	// Tanks
	{attribute 'OPC.UA.DA' := '1'}
  	{attribute 'OPC.UA.DA.StructuredType' := '1'}
	fbTank_PHUp: 		FB_Tank(TankID:= 'DTK1' ,TankDescr:= 'pH Up Nutrient Tank');
	{attribute 'OPC.UA.DA' := '1'}
  	{attribute 'OPC.UA.DA.StructuredType' := '1'} 
	fbTank_PHDown: 		FB_Tank(TankID:= 'DTK2' ,TankDescr:= 'pH Down Nutrient Tank');
	{attribute 'OPC.UA.DA' := '1'}
  	{attribute 'OPC.UA.DA.StructuredType' := '1'} 
	fbTank_NutrientA: 	FB_Tank(TankID:= 'DTK3' ,TankDescr:= 'Nutrient A Nutrient Tank');
	{attribute 'OPC.UA.DA' := '1'}
  	{attribute 'OPC.UA.DA.StructuredType' := '1'} 
	fbTank_NutrientB: 	FB_Tank(TankID:= 'DTK4' ,TankDescr:= 'Nutrient B Nutrient Tank');
	{attribute 'OPC.UA.DA' := '1'}
  	{attribute 'OPC.UA.DA.StructuredType' := '1'} 
	fbTank_NutrientC: 	FB_Tank(TankID:= 'DTK5' ,TankDescr:= 'Nutrient C Nutrient Tank'); 
	
	{attribute 'OPC.UA.DA' := '1'}
  	{attribute 'OPC.UA.DA.StructuredType' := '1'}
	fbSensor_TankpHUP_LS1: 		FB_Sensor_SICKLevelSwitch_GRF18S(SensorID:= 'DTK1-LS1' , SensorDescr:= 'pH Up Level Switch', 	  SensorType:= E_SensorType.Digital);
	{attribute 'OPC.UA.DA' := '1'}
  	{attribute 'OPC.UA.DA.StructuredType' := '1'}
	fbSensor_TankpHDown_LS1: 	FB_Sensor_SICKLevelSwitch_GRF18S(SensorID:= 'DTK2-LS1' , SensorDescr:= 'pH Down Level Switch', 	  SensorType:= E_SensorType.Digital);
	{attribute 'OPC.UA.DA' := '1'}
  	{attribute 'OPC.UA.DA.StructuredType' := '1'}
	fbSensor_TankNutrientA_LS1: FB_Sensor_SICKLevelSwitch_GRF18S(SensorID:= 'DTK3-LS1' , SensorDescr:= 'Nutrient A Level Switch', SensorType:= E_SensorType.Digital);
	{attribute 'OPC.UA.DA' := '1'}
  	{attribute 'OPC.UA.DA.StructuredType' := '1'}
	fbSensor_TankNutrientB_LS1: FB_Sensor_SICKLevelSwitch_GRF18S(SensorID:= 'DTK4-LS1' , SensorDescr:= 'Nutrient B Level Switch', SensorType:= E_SensorType.Digital);
	{attribute 'OPC.UA.DA' := '1'}
  	{attribute 'OPC.UA.DA.StructuredType' := '1'}
	fbSensor_TankNutrientC_LS1: FB_Sensor_SICKLevelSwitch_GRF18S(SensorID:= 'DTK5-LS1' , SensorDescr:= 'Nutrient C Level Switch', SensorType:= E_SensorType.Digital);
	
	
	// Control Loops
	{attribute 'OPC.UA.DA' := '0'}
	fbControlLoop_Dosing: 		FB_ControlLoop_Dosing(
														DosingPump_phUp := fbDosingPump_phUp, 
														DosingPump_phDOwn := fbDosingPump_phDown, 
														DosingPump_Nutrient_A := fbDosingPump_NutrientA, 
														DosingPump_Nutrient_B := fbDosingPump_NutrientB, 
														DosingPump_Nutrient_C := fbDosingPump_NutrientC, 
														Sensor_EC := fbSensor_EC, 
														Sensor_DO := fbSensor_DissOx, 
														Sensor_ORP := fbSensor_ORP, 
														Sensor_PH := fbSensor_PH, 
														Sensor_TEMP := fbSensor_TMP);
														
	
													
	// Package all components into structure & array 
	// ST used for readability
	// Arrray used for iterability 
	{attribute 'OPC.UA.DA' := '0'}
	stAllComponents: ST_RNDDMComponents;
	
	
	// Interlocks
	{attribute 'OPC.UA.DA' := '1'}
  	{attribute 'OPC.UA.DA.StructuredType' := '1'}
	fbInterlocks: 		FB_InterlockManager;
	
	// Sequences
	{attribute 'OPC.UA.DA' := '0'}
	fbSeqRND_DMMain: 	FB_SequenceRND_Main;
	{attribute 'OPC.UA.DA' := '0'}
	fbSeqRND_DMCal: 	FB_SequenceRND_Calibrate;
	{attribute 'OPC.UA.DA' := '0'}
	fbSeqRND_DMFill: 	FB_SequenceRND_Fill;
	{attribute 'OPC.UA.DA' := '0'}
	aSeqs: ARRAY[1..5] OF FB_SequenceBase;
	
END_VAR

IF GVL.bAutoUpdateDeviceState THEN
	simulation();     // This auto-updates devices eState to the eStateTarget (for testing purposes only)
END_IF

IF bIsFirstRun  THEN
	devices_init();	
	sequence_init();
	bIsFirstRun := FALSE;
END_IF

scanOPCInputs(Inputs := stInputs );
fbSequenceManager(aSequences := aSeqs, fbCurrentSequence := aSeqs[1]);
fbControlLoop_Dosing();

IF GVL.bEnableInterlocks_DM THEN
	interlocks();
END_IF

devices_update();

METHOD checkWaterQuality : BOOL
VAR_INPUT
END_VAR
checkWaterQuality := TRUE;

IF fbSensor_DissOx.getValue() < nDO_Low_Limit OR
	fbSensor_DissOx.getValue() > nDO_High_Limit THEN
	
	checkWaterQuality := FALSE;
	// raise an event
END_IF

IF fbSensor_EC.getValue() < nEC_Low_Limit OR
	fbSensor_EC.getValue() > nEC_High_Limit THEN
	
	checkWaterQuality := FALSE;
	// raise an event
END_IF


IF fbSensor_ORP.getValue() < nORP_Low_Limit OR
	fbSensor_ORP.getValue() > nORP_High_Limit THEN
	
	checkWaterQuality := FALSE;
	// raise an event
END_IF


IF fbSensor_PH.getValue() < nPH_Low_Limit OR
	fbSensor_PH.getValue() > nPH_High_Limit THEN
	
	checkWaterQuality := FALSE;
	// raise an event
END_IF


IF fbSensor_TMP.getValue() < nTemp_Low_Limit OR
	fbSensor_TMP.getValue() > nTemp_High_Limit THEN
	
	checkWaterQuality := FALSE;
	// raise an event
END_IF
END_METHOD

METHOD devices_init : BOOL
VAR
	VarInfo : __SYSTEM.VAR_INFO;
END_VAR
// Hold References to devices in a structure and also an array
// A structure is useful where devices are accessed by name (handy with auto-complete and readability)
// The array is useful for when we want to iterate through all of the devices in the machine and apply a global command (i.e. disable all devices)

// Add physical entity sensors to physical entities (i.e. tanks)
fbSumpDosing.fbSensor_H := fbSensor_SumpLSH;
fbSumpDosing.bSensorH_Enable := TRUE;

fbTank_PHUp.fbSensor_H := fbSensor_TankpHUP_LS1;
fbTank_PHUp.bSensorH_Enable := TRUE;

fbTank_PHDown.fbSensor_H := fbSensor_TankpHDown_LS1;
fbTank_PHDown.bSensorH_Enable := TRUE;

fbTank_NutrientA.fbSensor_H := fbSensor_TankNutrientA_LS1;
fbTank_NutrientA.bSensorH_Enable := TRUE;

fbTank_NutrientB.fbSensor_H := fbSensor_TankNutrientB_LS1;
fbTank_NutrientB.bSensorH_Enable := TRUE;

fbTank_NutrientC.fbSensor_H := fbSensor_TankNutrientC_LS1;
fbTank_NutrientC.bSensorH_Enable := TRUE;

// Extract the function block instance name and insert it to each function block
// This enables us to share only the function block name over OPC for nested instances (i.e. sequences, interlock manager)
// The contents of each function block is shared over OPC within the Machine as per heirarchy
// When Ignition needs to retrieve details of devices at the interlock manager and sequence, it simply performs a lookup using the VarID as a key


VarInfo := __VARINFO(fbControlLoop_Dosing);
fbControlLoop_Dosing.setVarID(VarID := VarInfo.Symbol);

VarInfo := __VARINFO(fbDosingPump_NutrientA);
fbDosingPump_NutrientA.setVarID(VarID := VarInfo.Symbol);

VarInfo := __VARINFO(fbDosingPump_NutrientB);
fbDosingPump_NutrientB.setVarID(VarID := VarInfo.Symbol);

VarInfo := __VARINFO(fbDosingPump_NutrientC);
fbDosingPump_NutrientC.setVarID(VarID := VarInfo.Symbol);

VarInfo := __VARINFO(fbDosingPump_phDown);
fbDosingPump_phDown.setVarID(VarID := VarInfo.Symbol);

VarInfo := __VARINFO(fbDosingPump_phUp);
fbDosingPump_phUp.setVarID(VarID := VarInfo.Symbol);

VarInfo := __VARINFO(fbPump_MainPumpA);
fbPump_MainPumpA.setVarID(VarID := VarInfo.Symbol);

VarInfo := __VARINFO(fbSensor_DissOx);
fbSensor_DissOx.setVarID(VarID := VarInfo.Symbol);

VarInfo := __VARINFO(fbSensor_DosingPIT1);
fbSensor_DosingPIT1.setVarID(VarID := VarInfo.Symbol);

VarInfo := __VARINFO(fbSensor_EC);
fbSensor_EC.setVarID(VarID := VarInfo.Symbol);

VarInfo := __VARINFO(fbSensor_FilterPIT1);
fbSensor_FilterPIT1.setVarID(VarID := VarInfo.Symbol);

VarInfo := __VARINFO(fbSensor_FilterPIT2);
fbSensor_FilterPIT2.setVarID(VarID := VarInfo.Symbol);

VarInfo := __VARINFO(fbSensor_ORP);
fbSensor_ORP.setVarID(VarID := VarInfo.Symbol);

VarInfo := __VARINFO(fbSensor_PH);
fbSensor_PH.setVarID(VarID := VarInfo.Symbol);

VarInfo := __VARINFO(fbSensor_SumpLSH );
fbSensor_SumpLSH .setVarID(VarID := VarInfo.Symbol);

VarInfo := __VARINFO(fbSensor_TankNutrientA_LS1);
fbSensor_TankNutrientA_LS1.setVarID(VarID := VarInfo.Symbol);

VarInfo := __VARINFO(fbSensor_TankNutrientB_LS1);
fbSensor_TankNutrientB_LS1.setVarID(VarID := VarInfo.Symbol);

VarInfo := __VARINFO(fbSensor_TankNutrientC_LS1);
fbSensor_TankNutrientC_LS1.setVarID(VarID := VarInfo.Symbol);

VarInfo := __VARINFO(fbSensor_TankpHDown_LS1);
fbSensor_TankpHDown_LS1.setVarID(VarID := VarInfo.Symbol);

VarInfo := __VARINFO(fbSensor_TankpHUP_LS1);
fbSensor_TankpHUP_LS1.setVarID(VarID := VarInfo.Symbol);

VarInfo := __VARINFO(fbSensor_TMP);
fbSensor_TMP.setVarID(VarID := VarInfo.Symbol);

VarInfo := __VARINFO(fbSumpDosing);
fbSumpDosing.setVarID(VarID := VarInfo.Symbol);

VarInfo := __VARINFO(fbTank_NutrientA);
fbTank_NutrientA.setVarID(VarID := VarInfo.Symbol);

VarInfo := __VARINFO(fbTank_NutrientB);
fbTank_NutrientB.setVarID(VarID := VarInfo.Symbol);

VarInfo := __VARINFO(fbTank_NutrientC);
fbTank_NutrientC.setVarID(VarID := VarInfo.Symbol);

VarInfo := __VARINFO(fbTank_PHDown);
fbTank_PHDown.setVarID(VarID := VarInfo.Symbol);

VarInfo := __VARINFO(fbTank_PHUp);
fbTank_PHUp.setVarID(VarID := VarInfo.Symbol);

VarInfo := __VARINFO(fbUVFilter1);
fbUVFilter1.setVarID(VarID := VarInfo.Symbol);

VarInfo := __VARINFO(fbValve_IrrigatorSupply);
fbValve_IrrigatorSupply.setVarID(VarID := VarInfo.Symbol);

VarInfo := __VARINFO(fbValve_RevOsSupply);
fbValve_RevOsSupply.setVarID(VarID := VarInfo.Symbol);


aAllComponents[1]  :=  ADR(fbSensor_DissOx );
aAllComponents[2]  :=  ADR(fbSensor_EC );
aAllComponents[3]  :=  ADR(fbSensor_ORP );
aAllComponents[4]  :=  ADR(fbSensor_PH );
aAllComponents[5]  :=  ADR(fbSensor_TMP );
aAllComponents[6]  :=  ADR(fbSensor_SumpLSH  );
aAllComponents[7]  :=  ADR(fbSensor_FilterPIT1 );
aAllComponents[8]  :=  ADR(fbSensor_FilterPIT2 );
aAllComponents[9]  :=  ADR(fbSensor_DosingPIT1 );
aAllComponents[10]  :=  ADR(fbDosingPump_phUp );
aAllComponents[11]  :=  ADR(fbDosingPump_phDown );
aAllComponents[12]  :=  ADR(fbDosingPump_NutrientA );
aAllComponents[13]  :=  ADR(fbDosingPump_NutrientB );
aAllComponents[14]  :=  ADR(fbDosingPump_NutrientC );
aAllComponents[15]  :=  ADR(fbValve_RevOsSupply );
aAllComponents[16]  :=  ADR(fbValve_IrrigatorSupply );
aAllComponents[17]  :=  ADR(fbPump_MainPumpA);
aAllComponents[18]  :=  ADR(fbUVFilter1 );
aAllComponents[19]  :=  ADR(fbSumpDosing );
aAllComponents[20]  :=  ADR(fbTank_PHUp );
aAllComponents[21]  :=  ADR(fbTank_PHDown );
aAllComponents[22]  :=  ADR(fbTank_NutrientA );
aAllComponents[23]  :=  ADR(fbTank_NutrientB );
aAllComponents[24]  :=  ADR(fbTank_NutrientC );
aAllComponents[25]  :=  ADR(fbSensor_TankpHUP_LS1 );
aAllComponents[26]  :=  ADR(fbSensor_TankpHDown_LS1 );
aAllComponents[27]  :=  ADR(fbSensor_TankNutrientA_LS1 );
aAllComponents[28]  :=  ADR(fbSensor_TankNutrientB_LS1 );
aAllComponents[29]  :=  ADR(fbSensor_TankNutrientC_LS1 );


stAllComponents.fbValve_RevOsSupply  := ADR(fbValve_RevOsSupply);
stAllComponents.fbValve_IrrigatorSupply  := ADR(fbValve_IrrigatorSupply);
stAllComponents.fbPump_MainPumpA  := ADR(fbPump_MainPumpA);
stAllComponents.fbUVFilter1  := ADR(fbUVFilter1);
stAllComponents.fbSumpDosing  := ADR(fbSumpDosing);
stAllComponents.fbDosingPump_phUp  := ADR(fbDosingPump_phUp);
stAllComponents.fbDosingPump_phDown  := ADR(fbDosingPump_phDown);
stAllComponents.fbDosingPump_NutrientA  := ADR(fbDosingPump_NutrientA);
stAllComponents.fbDosingPump_NutrientB  := ADR(fbDosingPump_NutrientB);
stAllComponents.fbDosingPump_NutrientC  := ADR(fbDosingPump_NutrientC);
stAllComponents.fbSensor_DissOx1  := ADR(fbSensor_DissOx);
stAllComponents.fbSensor_EC1  := ADR(fbSensor_EC);
stAllComponents.fbSensor_ORP1  := ADR(fbSensor_ORP);
stAllComponents.fbSensor_PH1  := ADR(fbSensor_PH);
stAllComponents.fbSensor_TMP1  := ADR(fbSensor_TMP);
stAllComponents.fbSensor_SumpLSH  := ADR(fbSensor_SumpLSH);
stAllComponents.fbSensor_TankpHUP_LS1  := ADR(fbSensor_TankpHUP_LS1);
stAllComponents.fbSensor_TankpHDown_LS1  := ADR(fbSensor_TankpHDown_LS1);
stAllComponents.fbSensor_TankNutrientA_LS1  := ADR(fbSensor_TankNutrientA_LS1);
stAllComponents.fbSensor_TankNutrientB_LS1  := ADR(fbSensor_TankNutrientB_LS1);
stAllComponents.fbSensor_TankNutrientC_LS1  := ADR(fbSensor_TankNutrientC_LS1);
stAllComponents.fbSensor_FilterPIT1  := ADR(fbSensor_FilterPIT1);
stAllComponents.fbSensor_FilterPIT2  := ADR(fbSensor_FilterPIT2);
stAllComponents.fbSensor_DosingPIT1  := ADR(fbSensor_DosingPIT1);
stAllComponents.fbTank_pHUP  := ADR(fbTank_pHUP);
stAllComponents.fbTank_pHDown  := ADR(fbTank_pHDown);
stAllComponents.fbTank_NutrientA  := ADR(fbTank_NutrientA);
stAllComponents.fbTank_NutrientB  := ADR(fbTank_NutrientB);
stAllComponents.fbTank_NutrientC  := ADR(fbTank_NutrientC);
stAllComponents.fbControlLoop_Dosing  := ADR(fbControlLoop_Dosing);

nQtyComponents := 29;

devices_disable_All();
END_METHOD

METHOD devices_update : BOOL
VAR_INPUT
END_VAR
fbModbusMaster();
fbDosingPump_phUp(fbModbusMaster := fbModbusMaster);
fbDosingPump_phDown(fbModbusMaster := fbModbusMaster);
fbDosingPump_NutrientA(fbModbusMaster := fbModbusMaster);
fbDosingPump_NutrientB(fbModbusMaster := fbModbusMaster);
fbDosingPump_NutrientC(fbModbusMaster := fbModbusMaster);
fbSensor_DissOx();
fbSensor_EC();
fbSensor_ORP();
fbSensor_PH();
fbSensor_TMP();
fbSensor_SumpLSH ();
fbSensor_FilterPIT1();
fbSensor_FilterPIT2();
fbSensor_DosingPIT1();
fbValve_RevOsSupply();
fbValve_IrrigatorSupply();
fbPump_MainPumpA();
fbUVFilter1();
fbSumpDosing();
fbTank_PHUp();
fbTank_PHDown();
fbTank_NutrientA();
fbTank_NutrientB();
fbTank_NutrientC();
fbSensor_TankpHUP_LS1();
fbSensor_TankpHDown_LS1();
fbSensor_TankNutrientA_LS1();
fbSensor_TankNutrientB_LS1();
fbSensor_TankNutrientC_LS1();
fbControlLoop_Dosing();
END_METHOD

METHOD FB_init : BOOL
VAR_INPUT
	bInitRetains : BOOL; // if TRUE, the retain variables are initialized (warm start / cold start)
	bInCopyCode : BOOL;  // if TRUE, the instance afterwards gets moved into the copy code (online change)
	
	ID: STRING;
	Description: STRING;
	//Pump_ModbusID: INT;
END_VAR
sID := ID;
sDescr := Description;
//nAgrowtekModbusID := Pump_ModbusID;
END_METHOD

METHOD interlocks : BOOL
VAR_INPUT
END_VAR
fbInterlocks.init();

fbInterlocks.update(
							Description:= 'Nutrient B Dosing Pump - RUNNING',
							InterlockType:= E_InterlockType.RunInterlock, 
							Subject_Device:= ADR(fbDosingPump_NutrientA), 
							Subject_State:= E_DeviceState.IDLE, 
							Signal:= E_DeviceState.RUNNING = fbDosingPump_NutrientB.getState(), 
							HoldSequence:=	TRUE );
				
							
fbInterlocks.update(
							Description:= 'Nutrient C Dosing Pump - RUNNING',
							InterlockType:= E_InterlockType.RunInterlock, 
							Subject_Device:= ADR(fbDosingPump_NutrientA), 
							Subject_State:= E_DeviceState.IDLE, 
							Signal:= fbDosingPump_NutrientC.getState() = E_DeviceState.RUNNING, 
							HoldSequence:=	TRUE );
							
fbInterlocks.update(
							Description:= 'PH Down Dosing Pump - RUNNING',
							InterlockType:= E_InterlockType.RunInterlock, 
							Subject_Device:= ADR(fbDosingPump_NutrientA), 
							Subject_State:= E_DeviceState.IDLE, 
							Signal := fbDosingPump_phDown.getState() = E_DeviceState.RUNNING, 
							HoldSequence:=	TRUE );
							
fbInterlocks.update(
							Description:= 'PH Up Dosing Pump - RUNNING',
							InterlockType:= E_InterlockType.RunInterlock, 
							Subject_Device:= ADR(fbDosingPump_NutrientA), 
							Subject_State:= E_DeviceState.IDLE, 
							Signal := fbDosingPump_phUp.getState() = E_DeviceState.RUNNING, 
							HoldSequence:=	TRUE );
								
							
fbInterlocks.update(
							Description:= 'Dosing Line Pressure - OUT OF RANGE',
							InterlockType:= E_InterlockType.RunInterlock, 
							Subject_Device:= ADR(fbDosingPump_NutrientA), 
							Subject_State:= E_DeviceState.IDLE, 
							Signal:= fbSensor_DosingPIT1.getState() = E_DeviceState.OUT_OF_RANGE, 
							HoldSequence:=	FALSE );
							
							
// Dosing Pump - Nutrient B Interlocks

fbInterlocks.update(
							Description:= 'Nutrient A Dosing Pump - RUNNING',
							InterlockType:= E_InterlockType.RunInterlock, 
							Subject_Device:= ADR(fbDosingPump_NutrientB), 
							Subject_State:= E_DeviceState.IDLE, 
							Signal:= fbDosingPump_NutrientA.getState() = E_DeviceState.RUNNING, 
							HoldSequence:=	TRUE );
							
fbInterlocks.update(
							Description:= 'Nutrient B Dosing Pump - RUNNING',
							InterlockType:= E_InterlockType.RunInterlock, 
							Subject_Device:= ADR(fbDosingPump_NutrientB), 
							Subject_State:= E_DeviceState.IDLE, 
							Signal := fbDosingPump_NutrientC.getState() = E_DeviceState.RUNNING, 
							HoldSequence:=	TRUE );
							
fbInterlocks.update(
							Description:= 'PH Down Dosing Pump - RUNNING',
							InterlockType:= E_InterlockType.RunInterlock, 
							Subject_Device:= ADR(fbDosingPump_NutrientB), 
							Subject_State:= E_DeviceState.IDLE, 
							Signal:= fbDosingPump_phDown.getState() = E_DeviceState.RUNNING, 
							HoldSequence:=	TRUE );
							
fbInterlocks.update(
							Description:= 'PH Up Dosing Pump - RUNNING',	
							InterlockType:= E_InterlockType.RunInterlock, 
							Subject_Device:= ADR(fbDosingPump_NutrientB), 
							Subject_State:= E_DeviceState.IDLE, 
							Signal:= fbDosingPump_phUp.getState() = E_DeviceState.RUNNING, 
							HoldSequence:=	TRUE );
							

							
fbInterlocks.update(
							Description:= 'Dosing Line Pressure - OUT OF RANGE',
							InterlockType:= E_InterlockType.RunInterlock, 
							Subject_Device:= ADR(fbDosingPump_NutrientB), 
							Subject_State:= E_DeviceState.IDLE, 
							Signal:= fbSensor_DosingPIT1.getState() = E_DeviceState.OUT_OF_RANGE, 
							HoldSequence:=	FALSE );

							
// Dosing Pump - Nutrient C Interlocks

fbInterlocks.update(
							Description:= 'Nutrient A Dosing Pump - RUNNING',
							InterlockType:= E_InterlockType.RunInterlock, 
							Subject_Device:= ADR(fbDosingPump_NutrientC), 
							Subject_State:= E_DeviceState.IDLE, 
							Signal:= fbDosingPump_NutrientA.getState() = E_DeviceState.RUNNING, 
							HoldSequence:=	TRUE );
							
fbInterlocks.update(
							Description:= 'Nutrient B Dosing Pump - RUNNING',
							InterlockType:= E_InterlockType.RunInterlock, 
							Subject_Device:= ADR(fbDosingPump_NutrientC), 
							Subject_State:= E_DeviceState.IDLE, 
							Signal:= fbDosingPump_NutrientB.getState() = E_DeviceState.RUNNING, 
							HoldSequence:=	TRUE );
							
fbInterlocks.update(
							Description:= 'PH Down Dosing Pump - RUNNING',	
							InterlockType:= E_InterlockType.RunInterlock, 
							Subject_Device:= ADR(fbDosingPump_NutrientC), 
							Subject_State:= E_DeviceState.IDLE, 
							Signal:= fbDosingPump_phDown.getState() = E_DeviceState.RUNNING, 
							HoldSequence:=	TRUE );
							
fbInterlocks.update(
							Description:= 'PH Up Dosing Pump - RUNNING',	
							InterlockType:= E_InterlockType.RunInterlock, 
							Subject_Device:= ADR(fbDosingPump_NutrientC), 
							Subject_State:= E_DeviceState.IDLE, 
							Signal:= fbDosingPump_phUp.getState() = E_DeviceState.RUNNING, 
							HoldSequence:=	TRUE );
							
							
fbInterlocks.update(
							Description:= 'Dosing Line Pressure - OUT OF RANGE',
							InterlockType:= E_InterlockType.StartPermissive, 
							Subject_Device:= ADR(fbDosingPump_NutrientC), 
							Subject_State:= E_DeviceState.IDLE, 
							Signal:= fbSensor_DosingPIT1.getState() = E_DeviceState.OUT_OF_RANGE, 
							HoldSequence:=	FALSE );
							
							
// Dosing Pump - PH Up Interlocks
fbInterlocks.update(
							Description:= 'Nutrient A Dosing Pump - RUNNING',	
							InterlockType:= E_InterlockType.RunInterlock, 
							Subject_Device:= ADR(fbDosingPump_phUp), 
							Subject_State:= E_DeviceState.IDLE, 
							Signal:= fbDosingPump_NutrientA.getState() = E_DeviceState.RUNNING, 
							HoldSequence:=	TRUE );
							
fbInterlocks.update(
							Description:= 'Nutrient B Dosing Pump - RUNNING',	
							InterlockType:= E_InterlockType.RunInterlock, 
							Subject_Device:= ADR(fbDosingPump_phUp), 
							Subject_State:= E_DeviceState.IDLE, 
							Signal:= fbDosingPump_NutrientB.getState() = E_DeviceState.RUNNING, 
							HoldSequence:=	TRUE );
							
fbInterlocks.update(
							Description:= 'Nutrient C Dosing Pump - RUNNING',
							InterlockType:= E_InterlockType.RunInterlock, 
							Subject_Device:= ADR(fbDosingPump_phUp), 
							Subject_State:= E_DeviceState.IDLE, 
							Signal:= fbDosingPump_NutrientC.getState() = E_DeviceState.RUNNING, 
							HoldSequence:=	TRUE );
							
fbInterlocks.update(
							Description:= 'PH Down Dosing Pump - RUNNING',
							InterlockType:= E_InterlockType.RunInterlock, 
							Subject_Device:= ADR(fbDosingPump_phUp), 
							Subject_State:= E_DeviceState.IDLE, 
							Signal:= fbDosingPump_phDown.getState() = E_DeviceState.RUNNING, 
							HoldSequence:=	TRUE );
					
							
fbInterlocks.update(
							Description:= 'Dosing Line Pressure - OUT OF RANGE',		
							InterlockType:= E_InterlockType.StartPermissive, 
							Subject_Device:= ADR(fbDosingPump_phUp), 
							Subject_State:= E_DeviceState.IDLE, 
							Signal:= fbSensor_DosingPIT1.getState() = E_DeviceState.OUT_OF_RANGE, 
							HoldSequence:=	FALSE );	
						
							
// Dosing Pump - PH Down Interlocks
fbInterlocks.update(
							Description:= 'Nutrient A Dosing Pump - RUNNING',		
							InterlockType:= E_InterlockType.RunInterlock, 
							Subject_Device:= ADR(fbDosingPump_phDown), 
							Subject_State:= E_DeviceState.IDLE, 
							Signal:= fbDosingPump_NutrientA.getState() = E_DeviceState.RUNNING, 
							HoldSequence:=	TRUE );
							
fbInterlocks.update(
							Description:= 'Nutrient B Dosing Pump - RUNNING',	
							InterlockType:= E_InterlockType.RunInterlock, 
							Subject_Device:= ADR(fbDosingPump_phDown), 
							Subject_State:= E_DeviceState.IDLE, 
							Signal:= fbDosingPump_NutrientB.getState() = E_DeviceState.RUNNING, 
							HoldSequence:=	TRUE );
							
fbInterlocks.update(
							Description:= 'Nutrient C Dosing Pump - RUNNING',	
							InterlockType:= E_InterlockType.RunInterlock, 
							Subject_Device:= ADR(fbDosingPump_phDown), 
							Subject_State:= E_DeviceState.IDLE, 
							Signal:= fbDosingPump_NutrientC.getState() = E_DeviceState.RUNNING, 
							HoldSequence:=	TRUE );
							
fbInterlocks.update(
							Description:= 'PH Up Dosing Pump - RUNNING',		
							InterlockType:= E_InterlockType.RunInterlock, 
							Subject_Device:= ADR(fbDosingPump_phDown), 
							Subject_State:= E_DeviceState.IDLE, 
							Signal:= fbDosingPump_phUp.getState() = E_DeviceState.RUNNING, 
							HoldSequence:=	TRUE );
							
fbInterlocks.update(
							Description:= 'Dosing Line Pressure - OUT OF RANGE',		
							InterlockType:= E_InterlockType.RunInterlock, 
							Subject_Device:= ADR(fbDosingPump_phDown), 
							Subject_State:= E_DeviceState.IDLE, 
							Signal:= fbSensor_DosingPIT1.getState() = E_DeviceState.OUT_OF_RANGE, 
							HoldSequence:=	FALSE );

							
// Main Pump A - Interlocks	
fbInterlocks.update(
							Description:= 'Dosing Sump - LOW LOW Level',	
							InterlockType:= E_InterlockType.RunInterlock, 
							Subject_Device:= ADR(fbPump_MainPumpA), 
							Subject_State:= E_DeviceState.IDLE, 
							Signal:= fbSumpDosing.getState() = E_DeviceState.LOW_LOW,
							HoldSequence:=	TRUE );	
										

							
							
							
fbInterlocks.update(
							Description:= 'Bag Filter 1 - OVER-PRESSURE',
							InterlockType:= E_InterlockType.RunInterlock, 
							Subject_Device:= ADR(fbPump_MainPumpA), 
							Subject_State:= E_DeviceState.IDLE, 
							Signal:= (fbSensor_FilterPIT2.getValue() - fbSensor_FilterPIT1.getValue())  > nBagFilterPressureMax,
							HoldSequence:=	TRUE ); 
							
fbInterlocks.update(
							Description:= 'Bag Filter 2 - OVER-PRESSURE',
							InterlockType:= E_InterlockType.RunInterlock, 
							Subject_Device:= ADR(fbPump_MainPumpA), 
							Subject_State:= E_DeviceState.IDLE, 
							Signal:= (fbSensor_DosingPIT1.getValue() - fbSensor_FilterPIT2.getValue()  > nBagFilterPressureMax),
							HoldSequence:=	TRUE );
	
							
// UV Filter - Interlocks					

fbInterlocks.update(
							Description:= 'Dosing Line - Low Pressure',
							InterlockType:= E_InterlockType.RunInterlock, 
							Subject_Device:= ADR(fbUVFilter1), 
							Subject_State:= E_DeviceState.OFF, 
							Signal:= fbSensor_DosingPIT1.getValue() < nPressureMin_Dosing, 
							HoldSequence:=	TRUE );	

// Valve - Irrigator Supply				

fbInterlocks.update(
							Description:= 'Water Quality (EC,pH,ORP,DO and temp) - OUT OF RANGE',
							InterlockType:= E_InterlockType.RunInterlock, 
							Subject_Device:= ADR(fbValve_IrrigatorSupply), 
							Subject_State:= E_DeviceState.CLOSED, 
							Signal:= checkWaterQuality(), 
							HoldSequence:=	TRUE );			
							
fbInterlocks.execute();
END_METHOD

METHOD scanOPCInputs : BOOL
VAR_INPUT
	Inputs: ST_INPUTS_RND_DosingMachine;
END_VAR

(*
			SEQUENCE CONTROL
*)



IF stInputs.stSequenceManager.Sequence_Selected <> fbSequenceManager.getCurrentSeq_ID() THEN // Selected sequence has been changed
	fbSequenceManager.stopSequence();
	devices_disable_All();
	fbSequenceManager.selectSequence(stInputs.stSequenceManager.Sequence_Selected);
	devices_enable_CurrSeq();
	//fbSequenceManager.startSequence(); // Automatically start sequence on change of sequence selected - can change this if required
END_IF


IF stInputs.stSequenceManager.Sequence_Ack_Interlock THEN
	fbSequenceManager.acknowledgePause();
	stInputs.stSequenceManager.Sequence_Ack_Interlock := FALSE;
END_IF



CASE stInputs.stSequenceManager.Sequence_Command OF
	E_SequenceState.RUN:
		IF fbSequenceManager.getState() <> E_SequenceState.RUN THEN
			fbSequenceManager.startSequence();
			stInputs.stSequenceManager.Sequence_Command := E_SequenceState.WAIT;
		END_IF
	E_SequenceState.STOP:
		IF fbSequenceManager.getState() <> E_SequenceState.STOP THEN
			fbSequenceManager.stopSequence();
			stInputs.stSequenceManager.Sequence_Command := E_SequenceState.WAIT;
		END_IF
	E_SequenceState.HOLD:
		IF fbSequenceManager.getState() <> E_SequenceState.HOLD THEN
			fbSequenceManager.pauseSequence();
			stInputs.stSequenceManager.Sequence_Command := E_SequenceState.WAIT;
		END_IF
END_CASE


(*
			WATER QUALITY LIMITS
*)


nEC_Low_Limit := stInputs.stWaterQuality.EC_LOW_Limit;
nEC_High_Limit := stInputs.stWaterQuality.EC_HIGH_Limit;
nEC_SetPoint := stInputs.stWaterQuality.EC_SetPoint;

nPH_Low_Limit := stInputs.stWaterQuality.PH_LOW_Limit;
nPH_High_Limit := stInputs.stWaterQuality.PH_HIGH_Limit;
nPH_SetPoint := stInputs.stWaterQuality.PH_SetPoint;

nDO_Low_Limit := stInputs.stWaterQuality.DO_LOW_Limit;
nDO_High_Limit := stInputs.stWaterQuality.DO_HIGH_Limit;
nDO_SetPoint := stInputs.stWaterQuality.DO_SetPoint;

nORP_Low_Limit := stInputs.stWaterQuality.ORP_LOW_Limit;
nORP_High_Limit := stInputs.stWaterQuality.ORP_HIGH_Limit;
nORP_SetPoint := stInputs.stWaterQuality.ORP_SetPoint;

nTemp_Low_Limit := stInputs.stWaterQuality.Temp_LOW_Limit;
nTemp_Low_Limit := stInputs.stWaterQuality.Temp_LOW_Limit;
nTemp_SetPoint := stInputs.stWaterQuality.Temp_SetPoint;

(*
			PRESSURE LIMITS
*)

//nPressureMin_Dosing := stInputs.Dosing_Pressure_LOW_Limit;
//nPressureMax_Dosing := stInputs.Dosing_Pressure_HIGH_Limit;


(*
			ACTUATORS
*)

fbValve_IrrigatorSupply.setMode(Mode := stInputs.stValve_IrrigatorSupply.Mode);
IF fbValve_IrrigatorSupply.inManual() THEN
	fbValve_IrrigatorSupply.setCommand(StateTarget := stInputs.stValve_IrrigatorSupply.Command);
END_IF

fbUVFilter1.setMode(Mode := stInputs.stUVFilter.Mode);
IF fbUVFilter1.inManual() THEN
	fbUVFilter1.setCommand(StateTarget := stInputs.stUVFilter.Command);
END_IF

// Dosing Pump - PH UP
fbDosingPump_phUp.setMode(Mode := stInputs.stDosingPump_phUp.Mode);
IF fbDosingPump_phUp.inManual() THEN
	fbDosingPump_phUp.setCommand(StateTarget := stInputs.stDosingPump_phUp.Command);
END_IF
						
// Dosing Pump - PH Down
fbDosingPump_phDown.setMode(Mode := stInputs.stDosingPump_phDown.Mode);
IF fbDosingPump_phDown.inManual() THEN
	fbDosingPump_phDown.setCommand(StateTarget := stInputs.stDosingPump_phDown.Command);
END_IF

// Dosing Pump - Nutrient A
fbDosingPump_NutrientA.setMode(Mode := stInputs.stDosingPump_NutrientA.Mode);
IF fbDosingPump_NutrientA.inManual() THEN
	fbDosingPump_NutrientA.setCommand(StateTarget := stInputs.stDosingPump_NutrientA.Command);
END_IF

// Dosing Pump - Nutrient B
fbDosingPump_NutrientB.setMode(Mode := stInputs.stDosingPump_NutrientB.Mode);
IF fbDosingPump_NutrientB.inManual() THEN
	fbDosingPump_NutrientB.setCommand(StateTarget := stInputs.stDosingPump_NutrientB.Command);
END_IF

// Dosing Pump - Nutrient C
fbDosingPump_NutrientC.setMode(Mode := stInputs.stDosingPump_NutrientC.Mode);
IF fbDosingPump_NutrientC.inManual() THEN
	fbDosingPump_NutrientC.setCommand(StateTarget := stInputs.stDosingPump_NutrientC.Command);
END_IF
						

// Main Pump A
fbPump_MainPumpA.setMode(Mode := stInputs.stPump_MainPumpA.Mode);
IF fbPump_MainPumpA.inManual() THEN
	fbPump_MainPumpA.setCommand(StateTarget := stInputs.stPump_MainPumpA.Command);
END_IF

// Control Loop						
fbControlLoop_Dosing.setParams(
								NutrientMaxDoseRate := stInputs.stControlLoopDosing_Nutrient.MaxDoseRate,
								NutrientMinDoseRate := stInputs.stControlLoopDosing_Nutrient.MinDoseRate,
								NutrientTimeBetweenDoses := UINT_TO_TIME(stInputs.stControlLoopDosing_Nutrient.TimeBetweenDoses),
								
								// VAR_INPUTS
								NutrientSetpoint  := stInputs.stControlLoopDosing_Nutrient.Setpoint,
								NutrientManSyncVal  := stInputs.stControlLoopDosing_Nutrient.ManSyncVal,
								NutrientSync  := stInputs.stControlLoopDosing_Nutrient.Sync,
								NutrientMode  := stInputs.stControlLoopDosing_Nutrient.Mode,
								NutrientHold  := stInputs.stControlLoopDosing_Nutrient.Hold,
								
								// VAR_IN_OUT (ST_PARAMS)
								NutrientCtrlCycleTime  := UINT_TO_TIME(stInputs.stControlLoopDosing_Nutrient.CtrlCycleTime),
								NutrientTaskCycleTime  := UINT_TO_TIME(stInputs.stControlLoopDosing_Nutrient.TaskCycleTime),
								NutrientKp  := stInputs.stControlLoopDosing_Nutrient.Kp,
								NutrientTn  := UINT_TO_TIME(stInputs.stControlLoopDosing_Nutrient.Tn),
								NutrientTv  := UINT_TO_TIME(stInputs.stControlLoopDosing_Nutrient.Tv),
								NutrientTd  := UINT_TO_TIME(stInputs.stControlLoopDosing_Nutrient.Td),
								NutrientOutMaxLimit  := stInputs.stControlLoopDosing_Nutrient.OutMaxLimit,
								NutrientOutMinLimit  := stInputs.stControlLoopDosing_Nutrient.OutMinLimit,
								NutrientPInTheFeedbackPath := stInputs.stControlLoopDosing_Nutrient.PInTheFeedbackPath,
								NutrientDInTheFeedbackPath := stInputs.stControlLoopDosing_Nutrient.DInTheFeedbackPath,
								NutrientARWOnIPartOnly  := stInputs.stControlLoopDosing_Nutrient.ARWOnIPartOnly,
								
								NutrientSetpointBand  := stInputs.stControlLoopDosing_Nutrient.SetpointBand,
								
								PHMaxDoseRate := stInputs.stControlLoopDosing_PH.MaxDoseRate,
								PHMinDoseRate := stInputs.stControlLoopDosing_PH.MinDoseRate,
								PHTimeBetweenDoses := UINT_TO_TIME(stInputs.stControlLoopDosing_PH.TimeBetweenDoses),
								
								// VAR_INPUTS
								PHSetpoint  := stInputs.stControlLoopDosing_PH.Setpoint,
								PHManSyncVal  := stInputs.stControlLoopDosing_PH.ManSyncVal,
								PHSync  := stInputs.stControlLoopDosing_PH.Sync,
								PHMode  := stInputs.stControlLoopDosing_PH.Mode,
								PHHold  := stInputs.stControlLoopDosing_PH.Hold,
								
								// VAR_IN_OUT (ST_PARAMS)
								PHCtrlCycleTime  := UINT_TO_TIME(stInputs.stControlLoopDosing_PH.CtrlCycleTime),
								PHTaskCycleTime  := UINT_TO_TIME(stInputs.stControlLoopDosing_PH.TaskCycleTime),
								PHKp  := stInputs.stControlLoopDosing_PH.Kp,
								PHTn  := UINT_TO_TIME(stInputs.stControlLoopDosing_PH.Tn),
								PHTv  := UINT_TO_TIME(stInputs.stControlLoopDosing_PH.Tv),
								PHTd  := UINT_TO_TIME(stInputs.stControlLoopDosing_PH.Td),
								PHOutMaxLimit  := stInputs.stControlLoopDosing_PH.OutMaxLimit,
								PHOutMinLimit  := stInputs.stControlLoopDosing_PH.OutMinLimit,
								PHPInTheFeedbackPath  := stInputs.stControlLoopDosing_PH.PInTheFeedbackPath,
								PHDInTheFeedbackPath  := stInputs.stControlLoopDosing_PH.DInTheFeedbackPath,
								PHARWOnIPartOnly  := stInputs.stControlLoopDosing_PH.ARWOnIPartOnly,

								PHSetpointBand  := stInputs.stControlLoopDosing_PH.SetpointBand);
END_METHOD

METHOD sequence_init : BOOL
VAR_INPUT
END_VAR
fbSeqRND_DMMain(devices := stAllComponents);
fbSeqRND_DMCal(devices := stAllComponents);
fbSeqRND_DMFill(devices := stAllComponents);

fbSeqRND_DMMain.populateSteps();
fbSeqRND_DMCal.populateSteps();
fbSeqRND_DMFill.populateSteps();

aSeqs[1] := fbSeqRND_DMMain;
aSeqs[2] := fbSeqRND_DMCal;
aSeqs[3] := fbSeqRND_DMFill;
END_METHOD

METHOD simulation : BOOL
VAR_INPUT
END_VAR
END_METHOD

METHOD updateInputs : BOOL
VAR_INPUT
END_VAR
END_METHOD

END_FUNCTION_BLOCK

// ---- POUs/07 Systems/RND/FB_System_RND_GasMonitoring.TcPOU
FUNCTION_BLOCK FB_System_RND_GasMonitoring
VAR_IN_OUT
	// Hold a reference to MBMaster - may need to share this with other dosing machines if only 1 x RS485 card is used for both
	{attribute 'OPC.UA.DA' := '0'}
	fbModbusMaster_1: 	FB_ModbusMaster;
	fbModbusMaster_2: 	FB_ModbusMaster;    
END_VAR

VAR
	bFirstRun: BOOL := TRUE;
	
	eSMState: (O2_CONC, O2_AL1, O2_AL2, O2_AL3, CO2_CONC, CO2_AL1, CO2_AL2, CO2_AL3);
	
	nIterator: UINT := 1;
	
	{attribute 'OPC.UA.DA' := '1'}
  	{attribute 'OPC.UA.DA.StructuredType' := '1'}
	fbRND1_GAS: FB_GasMonitoringPanel_CDA4022(ModbusID:= GVL.RND1_GasMon_ModID);
	{attribute 'OPC.UA.DA' := '1'}
  	{attribute 'OPC.UA.DA.StructuredType' := '1'}
	fbRND2_GAS: FB_GasMonitoringPanel_CDA4022(ModbusID:= GVL.RND2_GasMon_ModID);
	{attribute 'OPC.UA.DA' := '1'}
  	{attribute 'OPC.UA.DA.StructuredType' := '1'}
	fbRND3_GAS: FB_GasMonitoringPanel_CDA4022(ModbusID:= GVL.RND3_GasMon_ModID);
	{attribute 'OPC.UA.DA' := '1'}
  	{attribute 'OPC.UA.DA.StructuredType' := '1'}
	fbRND4_GAS: FB_GasMonitoringPanel_CDA4022(ModbusID:= GVL.RND4_GasMon_ModID);
	{attribute 'OPC.UA.DA' := '1'}
  	{attribute 'OPC.UA.DA.StructuredType' := '1'}
	fbRND5_GAS: FB_GasMonitoringPanel_CDA4022(ModbusID:= GVL.RND5_GasMon_ModID);
	{attribute 'OPC.UA.DA' := '1'}
  	{attribute 'OPC.UA.DA.StructuredType' := '1'}
	fbRND6_GAS: FB_GasMonitoringPanel_CDA4022(ModbusID:= GVL.RND6_GasMon_ModID);
	{attribute 'OPC.UA.DA' := '1'}
  	{attribute 'OPC.UA.DA.StructuredType' := '1'}
	fbRND7_GAS: FB_GasMonitoringPanel_CDA4022(ModbusID:= GVL.RND7_GasMon_ModID);
	{attribute 'OPC.UA.DA' := '1'}
  	{attribute 'OPC.UA.DA.StructuredType' := '1'}
	fbRND8_GAS: FB_GasMonitoringPanel_CDA4022(ModbusID:= GVL.RND8_GasMon_ModID);
	{attribute 'OPC.UA.DA' := '1'}
  	{attribute 'OPC.UA.DA.StructuredType' := '1'}
	fbRND9_GAS: FB_GasMonitoringPanel_CDA4022(ModbusID:= GVL.RND9_GasMon_ModID);
	{attribute 'OPC.UA.DA' := '1'}
  	{attribute 'OPC.UA.DA.StructuredType' := '1'}
	fbRND10_GAS: FB_GasMonitoringPanel_CDA4022(ModbusID:= GVL.RND10_GasMon_ModID);
	{attribute 'OPC.UA.DA' := '1'}
  	{attribute 'OPC.UA.DA.StructuredType' := '1'}
	fbRND11_GAS: FB_GasMonitoringPanel_CDA4022(ModbusID:= GVL.RND11_GasMon_ModID);
	{attribute 'OPC.UA.DA' := '1'}
  	{attribute 'OPC.UA.DA.StructuredType' := '1'}
	fbRND12_GAS: FB_GasMonitoringPanel_CDA4022(ModbusID:= GVL.RND12_GasMon_ModID);
	
	aGasPanels: ARRAY[1..12] OF POINTER TO FB_GasMonitoringPanel_CDA4022;
END_VAR

IF bFirstRun THEN
	devices_init();
	bFirstRun := FALSE;
END_IF

devices_update();

CASE eSMState OF
	
	O2_CONC:
		IF aGasPanels[nIterator]^.read_Concentration_O2() THEN
			eSMState := O2_AL1;
		END_IF
		
	O2_AL1:
		IF aGasPanels[nIterator]^.read_Alarm_O2_Lvl1() THEN
			eSMState := O2_AL2;
		END_IF
		
	O2_AL2:
		IF aGasPanels[nIterator]^.read_Alarm_O2_Lvl2() THEN
			eSMState := O2_AL3;
		END_IF
		
	O2_AL3:
		IF aGasPanels[nIterator]^.read_Alarm_O2_Lvl3() THEN
			eSMState := CO2_CONC;
		END_IF
		
	CO2_CONC:
		IF aGasPanels[nIterator]^.read_Concentration_CO2() THEN
			eSMState := CO2_AL1;
		END_IF
		
	CO2_AL1:
		IF aGasPanels[nIterator]^.read_Alarm_CO2_Lvl1() THEN
			eSMState := CO2_AL2;
		END_IF
		
	CO2_AL2:
		IF aGasPanels[nIterator]^.read_Alarm_CO2_Lvl2() THEN
			eSMState := CO2_AL3;
		END_IF
		
	CO2_AL3:
		IF aGasPanels[nIterator]^.read_Alarm_CO2_Lvl3() THEN
			eSMState := O2_CONC;
			nIterator := nIterator + 1;
			IF nIterator > 12 THEN
				nIterator := 1;
			END_IF
		END_IF
	
END_CASE

METHOD devices_init : BOOL
VAR_INPUT
END_VAR

aGasPanels[1] := ADR(fbRND1_GAS);
aGasPanels[2] := ADR(fbRND2_GAS);
aGasPanels[3] := ADR(fbRND3_GAS);
aGasPanels[4] := ADR(fbRND4_GAS);
aGasPanels[5] := ADR(fbRND5_GAS);
aGasPanels[6] := ADR(fbRND6_GAS);
aGasPanels[7] := ADR(fbRND7_GAS);
aGasPanels[8] := ADR(fbRND8_GAS);
aGasPanels[9] := ADR(fbRND9_GAS);
aGasPanels[10] := ADR(fbRND10_GAS);
aGasPanels[11] := ADR(fbRND11_GAS);
aGasPanels[12] := ADR(fbRND12_GAS);
END_METHOD

METHOD devices_update : BOOL
VAR_INPUT
END_VAR
fbRND1_GAS(fbModbusMaster := fbModbusMaster_1);
fbRND2_GAS(fbModbusMaster := fbModbusMaster_1);
fbRND3_GAS(fbModbusMaster := fbModbusMaster_1);
fbRND4_GAS(fbModbusMaster := fbModbusMaster_1);
fbRND5_GAS(fbModbusMaster := fbModbusMaster_1);
fbRND6_GAS(fbModbusMaster := fbModbusMaster_1);

fbRND7_GAS(fbModbusMaster := fbModbusMaster_2);
fbRND8_GAS(fbModbusMaster := fbModbusMaster_2);
fbRND9_GAS(fbModbusMaster := fbModbusMaster_2);
fbRND10_GAS(fbModbusMaster := fbModbusMaster_2);
fbRND11_GAS(fbModbusMaster := fbModbusMaster_2);
fbRND12_GAS(fbModbusMaster := fbModbusMaster_2);
END_METHOD

END_FUNCTION_BLOCK

// ---- POUs/07 Systems/RND/FB_System_RND_GasMonitoring_R2.TcPOU
FUNCTION_BLOCK FB_System_RND_GasMonitoring_R2
VAR_IN_OUT
	// Hold a reference to MBMaster - may need to share this with other dosing machines if only 1 x RS485 card is used for both
	{attribute 'OPC.UA.DA' := '0'}
	fbModbusManager_1: 	FB_ModbusManager;
	fbModbusManager_2: 	FB_ModbusManager;    
END_VAR

VAR
	bFirstRun: BOOL := TRUE;
	
	eSMState: (O2_CONC, O2_AL1, O2_AL2, O2_AL3, CO2_CONC, CO2_AL1, CO2_AL2, CO2_AL3);
	
	nIterator: UINT := 1;
	
	{attribute 'OPC.UA.DA' := '1'}
  	{attribute 'OPC.UA.DA.StructuredType' := '1'}
	fbRND1_GAS: FB_GasMonitoringPanel_CDA4022_R2(ModbusID:= GVL.RND1_GasMon_ModID);
	{attribute 'OPC.UA.DA' := '1'}
  	{attribute 'OPC.UA.DA.StructuredType' := '1'}
	fbRND2_GAS: FB_GasMonitoringPanel_CDA4022_R2(ModbusID:= GVL.RND2_GasMon_ModID);
	{attribute 'OPC.UA.DA' := '1'}
  	{attribute 'OPC.UA.DA.StructuredType' := '1'}
	fbRND3_GAS: FB_GasMonitoringPanel_CDA4022_R2(ModbusID:= GVL.RND3_GasMon_ModID);
	{attribute 'OPC.UA.DA' := '1'}
  	{attribute 'OPC.UA.DA.StructuredType' := '1'}
	fbRND4_GAS: FB_GasMonitoringPanel_CDA4022_R2(ModbusID:= GVL.RND4_GasMon_ModID);
	{attribute 'OPC.UA.DA' := '1'}
  	{attribute 'OPC.UA.DA.StructuredType' := '1'}
	fbRND5_GAS: FB_GasMonitoringPanel_CDA4022_R2(ModbusID:= GVL.RND5_GasMon_ModID);
	{attribute 'OPC.UA.DA' := '1'}
  	{attribute 'OPC.UA.DA.StructuredType' := '1'}
	fbRND6_GAS: FB_GasMonitoringPanel_CDA4022_R2(ModbusID:= GVL.RND6_GasMon_ModID);
	{attribute 'OPC.UA.DA' := '1'}
  	{attribute 'OPC.UA.DA.StructuredType' := '1'}
	fbRND7_GAS: FB_GasMonitoringPanel_CDA4022_R2(ModbusID:= GVL.RND7_GasMon_ModID);
	{attribute 'OPC.UA.DA' := '1'}
  	{attribute 'OPC.UA.DA.StructuredType' := '1'}
	fbRND8_GAS: FB_GasMonitoringPanel_CDA4022_R2(ModbusID:= GVL.RND8_GasMon_ModID);
	{attribute 'OPC.UA.DA' := '1'}
  	{attribute 'OPC.UA.DA.StructuredType' := '1'}
	fbRND9_GAS: FB_GasMonitoringPanel_CDA4022_R2(ModbusID:= GVL.RND9_GasMon_ModID);
	{attribute 'OPC.UA.DA' := '1'}
  	{attribute 'OPC.UA.DA.StructuredType' := '1'}
	fbRND10_GAS: FB_GasMonitoringPanel_CDA4022_R2(ModbusID:= GVL.RND10_GasMon_ModID);
	{attribute 'OPC.UA.DA' := '1'}
  	{attribute 'OPC.UA.DA.StructuredType' := '1'}
	fbRND11_GAS: FB_GasMonitoringPanel_CDA4022_R2(ModbusID:= GVL.RND11_GasMon_ModID);
	{attribute 'OPC.UA.DA' := '1'}
  	{attribute 'OPC.UA.DA.StructuredType' := '1'}
	fbRND12_GAS: FB_GasMonitoringPanel_CDA4022_R2(ModbusID:= GVL.RND12_GasMon_ModID);
	
	aGasPanels: ARRAY[1..12] OF POINTER TO FB_GasMonitoringPanel_CDA4022_R2;
END_VAR

IF bFirstRun THEN
	devices_init();
	bFirstRun := FALSE;
END_IF

devices_update();

METHOD devices_init : BOOL
VAR_INPUT
END_VAR

aGasPanels[1] := ADR(fbRND1_GAS);
aGasPanels[2] := ADR(fbRND2_GAS);
aGasPanels[3] := ADR(fbRND3_GAS);
aGasPanels[4] := ADR(fbRND4_GAS);
aGasPanels[5] := ADR(fbRND5_GAS);
aGasPanels[6] := ADR(fbRND6_GAS);
aGasPanels[7] := ADR(fbRND7_GAS);
aGasPanels[8] := ADR(fbRND8_GAS);
aGasPanels[9] := ADR(fbRND9_GAS);
aGasPanels[10] := ADR(fbRND10_GAS);
aGasPanels[11] := ADR(fbRND11_GAS);
aGasPanels[12] := ADR(fbRND12_GAS);
END_METHOD

METHOD devices_update : BOOL
VAR_INPUT
END_VAR
fbRND1_GAS(fbModbusManager := fbModbusManager_1);
fbRND2_GAS(fbModbusManager := fbModbusManager_1);
fbRND3_GAS(fbModbusManager := fbModbusManager_1);
fbRND4_GAS(fbModbusManager := fbModbusManager_1);
fbRND5_GAS(fbModbusManager := fbModbusManager_1);
fbRND6_GAS(fbModbusManager := fbModbusManager_1);

fbRND7_GAS(fbModbusManager := fbModbusManager_2);
fbRND8_GAS(fbModbusManager := fbModbusManager_2);
fbRND9_GAS(fbModbusManager := fbModbusManager_2);
fbRND10_GAS(fbModbusManager := fbModbusManager_2);
fbRND11_GAS(fbModbusManager := fbModbusManager_2);
fbRND12_GAS(fbModbusManager := fbModbusManager_2);
END_METHOD

END_FUNCTION_BLOCK

// ---- POUs/99 Utilities/FB_HealthMonitoring.TcPOU
FUNCTION_BLOCK FB_HealthMonitoring EXTENDS FB_BaseDevice
VAR_INPUT
	fbTON_On_OFF: TON := (PT:= T#1S);
	
	{attribute 'OPC.UA.DA' := '1'}
	bHeartBeat: BOOL := FALSE;
	
	bResetTimer: BOOL := TRUE;
	
	nQtyCardStatus: INT := 40;
	
	aCardStatus: ARRAY[1..1000] OF BOOL;
	
	
END_VAR

IF bResetTimer THEN
	fbTON_On_OFF(IN := TRUE);
END_IF

IF fbTON_On_OFF.Q THEN
	bHeartBeat := (NOT bHeartBeat);
	fbTON_On_OFF(IN := FALSE);
	bResetTimer := TRUE;
END_IF

END_FUNCTION_BLOCK

// ---- POUs/99 Utilities/FB_RS485_CardRead.TcPOU
FUNCTION_BLOCK FB_RS485_CardRead

VAR
	fbSDORead: FB_EcCoeSdoRead;
	
	// Inputs
	sNetID: 		T_AmsNetId := '192.168.1.31.2.1'; 	// This is a string that contains the AMS network identifier of the EtherCAT master device.
	nSlaveAddr: 	UINT := 1005; 						// Fixed address of the EtherCAT slave to which the SDO upload command should be sent.
	nSubIndex:		BYTE; 								// Sub-index of the object that is to be read.
	nIndex:			WORD := 16#8000;								// Index of the object that is to be read.
	//pDstBuf:		DWORD; 								// The address (pointer) of the receive buffer
	rxBuffer:		ARRAY[1..16] OF BYTE;
	cbBufLen: 		UDINT; 								// The maximum available buffer size for the data to be read, in bytes.
	bExecute: 		BOOL; 								// The block is activated by a rising edge at this input.
	tTimeout:		TIME:=DEFAULT_ADS_TIMEOUT;
	
	// Outputs
	bBusy: 			BOOL; // This output is set when the function block is activated and remains set until an acknowledgement is received.
	bError:			BOOL; // This output is set up after the bBusy output has been reset if there has been an error in transmission of the command.
	nErrId:			UDINT; // Supplies the ADS error code associated with the most recently executed command if the bError output is set.
	
	

END_VAR

fbSdoRead();

METHOD readBaudrate : BOOL
VAR_OUTPUT
	Baudrate: POINTER TO DINT;
END_VAR
nSubIndex 	:= 16#11;
nIndex 		:= 16#8000;

fbSdoRead(sNetId:=sNetId, nSlaveAddr:=nSlaveAddr, nIndex:=nIndex, nSubIndex:=nSubIndex, pDstBuf:=Baudrate, cbBufLen:=SIZEOF(Baudrate^), bExecute:=bExecute);
bError:=fbSdoRead.bError;
nErrId:=fbSdoRead.nErrId;
bExecute := FALSE;
END_METHOD

METHOD readDataFrame : BOOL
VAR_INPUT
	Dataframe: POINTER TO INT;
END_VAR
nSubIndex 	:= 16#11;
nIndex 		:= 16#8000;

fbSdoRead(sNetId:=sNetId, nSlaveAddr:=nSlaveAddr, nIndex:=nIndex, nSubIndex:=nSubIndex, pDstBuf:=Dataframe, cbBufLen:=SIZEOF(Dataframe^), bExecute:=bExecute);
bError:=fbSdoRead.bError;
nErrId:=fbSdoRead.nErrId;
bExecute := FALSE;
END_METHOD

METHOD readInitAccepted : BOOL
VAR_INPUT
	Accepted: POINTER TO BOOL;
END_VAR
nSubIndex 	:= 16#3;
nIndex 		:= 16#6010;

fbSdoRead(sNetId:=sNetId, nSlaveAddr:=nSlaveAddr, nIndex:=nIndex, nSubIndex:=nSubIndex, pDstBuf:=Accepted, cbBufLen:=SIZEOF(Accepted^), bExecute:=bExecute);
bError:=fbSdoRead.bError;
nErrId:=fbSdoRead.nErrId;
bExecute := FALSE;
END_METHOD

METHOD readTxAccepted : BOOL
VAR_INPUT
	Accepted: POINTER TO BOOL;
END_VAR
nSubIndex 	:= 16#1;
nIndex 		:= 16#6010;

fbSdoRead(sNetId:=sNetId, nSlaveAddr:=nSlaveAddr, nIndex:=nIndex, nSubIndex:=nSubIndex, pDstBuf:=Accepted, cbBufLen:=SIZEOF(Accepted^), bExecute:=bExecute);
bError:=fbSdoRead.bError;
nErrId:=fbSdoRead.nErrId;
bExecute := FALSE;
END_METHOD

METHOD SDO_Read : BOOL
VAR_INPUT
END_VAR
END_METHOD

END_FUNCTION_BLOCK

// ---- POUs/99 Utilities/FB_RS485_CardWrite.TcPOU
FUNCTION_BLOCK FB_RS485_CardWrite

VAR
	fbSdoWrite: FB_EcCoESdoWrite;
	
	// Inputs
	sNetID: 		T_AmsNetId := '192.168.1.31.2.1'; 	// This is a string that contains the AMS network identifier of the EtherCAT master device.
	nSlaveAddr: 	UINT := 1005; 						// Fixed address of the EtherCAT slave to which the SDO upload command should be sent.
	nSubIndex:		BYTE := 16#11;								// Sub-index of the object that is to be read.
	nIndex:			WORD := 16#8000;								// Index of the object that is to be read.
	//pDstBuf:		DWORD; 								// The address (pointer) of the receive buffer
	nValue:			BYTE;
	cbBufLen: 		UDINT; 								// The maximum available buffer size for the data to be read, in bytes.
	bExecute: 		BOOL; 								// The block is activated by a rising edge at this input.
	tTimeout:		TIME := DEFAULT_ADS_TIMEOUT;
	
	// Outputs
	bBusy: 			BOOL; // This output is set when the function block is activated and remains set until an acknowledgement is received.
	bError:			BOOL; // This output is set up after the bBusy output has been reset if there has been an error in transmission of the command.
	nErrId:			UDINT; // Supplies the ADS error code associated with the most recently executed command if the bError output is set.
	
	
	bBool: BOOL := TRUE;
	
	// Index 16#8000 Sub 16#11 for Baudrate (7 - 19,200, 8 - 38,400) - use Byte type
	// Index 16#8000 Sub 16#15 for Baudrate (3 - 8N1, 11 - 8N2) 

END_VAR

(* fbSdoRead(sNetId:=sNetId, nSlaveAddr:=nSlaveAddr, nIndex:=nIndex, nSubIndex:=nSubIndex, pDstBuf:=ADR(rxBuffer), cbBufLen:=SIZEOF(rxBuffer), bExecute:=bExecute);
bError:=fbSdoRead.bError;
nErrId:=fbSdoRead.nErrId;
bExecute := FALSE;
*)


fbSdoWrite();

IF NOT fbSdoWrite.bBusy THEN
	bExecute:=FALSE;
IF NOT bError THEN
	(* write successful *)
	bError := FALSE;
	nErrId := 0;
ELSE
	(* write failed *)
	bError := fbSdoWrite.bError;
	nErrId := fbSdoWrite.nErrId;
END_IF
	fbSdoWrite(bExecute:=FALSE);
END_IF

METHOD isBusy : BOOL
VAR_INPUT
END_VAR
IF bBusy THEN
	isBusy := TRUE;
ELSE
	isBusy := FALSE;
END_IF
END_METHOD

METHOD writeBaud : BOOL
VAR_INPUT
	Baudrate: DINT;
END_VAR
IF NOT bBusy THEN
	nIndex := 16#8000;
	nSubIndex := 16#11;
	
	CASE Baudrate OF
		300:
			nValue := 1;
		600:
			nValue := 2;
		1200:
			nValue := 3;
		2400:
			nValue := 4;
		4800:
			nValue := 5;
		9600:
			nValue := 6;
		19200:
			nValue := 7;
		38400:
			nValue := 8;
		57600:
			nValue := 9;
		115200:
			nValue := 9;
	END_CASE
	
	bExecute := TRUE;
	
	fbSdoWrite(
			sNetId :=		sNetId,
			nSlaveAddr :=	nSlaveAddr,
			nIndex :=		nIndex,
			nSubIndex :=	nSubIndex,
			pSrcBuf :=		ADR(nValue),
			cbBufLen :=		SIZEOF(nValue),
			bExecute :=		bExecute
);
	writeBaud := TRUE;
ELSE
	writeBaud := FALSE;
	
END_IF
END_METHOD

METHOD writeDataFrame : BOOL
VAR_INPUT
	Dataframe: STRING;
END_VAR
IF NOT bBusy THEN
	nIndex := 16#8000;
	nSubIndex := 16#15;
	
	IF Dataframe = '7E1' THEN
		nValue := 1;
	ELSIF Dataframe = '7O1' THEN
		nValue := 2;
	ELSIF Dataframe = '8N1' THEN
		nValue := 2;
	ELSIF Dataframe = '8E1' THEN
		nValue := 2;
	ELSIF Dataframe = '8O1' THEN
		nValue := 2;
	ELSIF Dataframe = '7E2' THEN
		nValue := 2;
	ELSIF Dataframe = '7O2' THEN
		nValue := 2;
	ELSIF Dataframe = '8N2' THEN
		nValue := 2;
	ELSIF Dataframe = '8E2' THEN
		nValue := 2;
	ELSIF Dataframe = '8O2' THEN
		nValue := 2;
	ELSE
		writeDataFrame := FALSE;
	END_IF

	bExecute := TRUE;
	
	fbSdoWrite(
			sNetId :=		sNetId,
			nSlaveAddr :=	nSlaveAddr,
			nIndex :=		nIndex,
			nSubIndex :=	nSubIndex,
			pSrcBuf :=		ADR(nValue),
			cbBufLen :=		SIZEOF(nValue),
			bExecute :=		bExecute
	);
	writeDataFrame := TRUE;
ELSE
	writeDataFrame := FALSE;
	
END_IF
END_METHOD

METHOD writeInitRequest : BOOL
VAR_INPUT
END_VAR
IF NOT bBusy THEN
	nIndex := 16#7000;
	nSubIndex := 16#3;
	bBool := TRUE;
	bExecute := TRUE;
	
	fbSdoWrite(
			sNetId :=		sNetId,
			nSlaveAddr :=	nSlaveAddr,
			nIndex :=		nIndex,
			nSubIndex :=	nSubIndex,
			pSrcBuf :=		ADR(bBool),
			cbBufLen :=		SIZEOF(bBool),
			bExecute :=		bExecute
	);
	writeInitRequest := TRUE;
ELSE
	writeInitRequest := FALSE;
END_IF
END_METHOD

METHOD writeTxRequest : BOOL
VAR_INPUT
END_VAR
IF NOT bBusy THEN
	nIndex := 16#7000;
	nSubIndex := 16#1;
	bBool := TRUE;
	bExecute := TRUE;
	
	fbSdoWrite(
			sNetId :=		sNetId,
			nSlaveAddr :=	nSlaveAddr,
			nIndex :=		nIndex,
			nSubIndex :=	nSubIndex,
			pSrcBuf :=		ADR(bBool),
			cbBufLen :=		SIZEOF(bBool),
			bExecute :=		bExecute
	);
	writeTxRequest := TRUE;
ELSE
	writeTxRequest := FALSE;
END_IF
END_METHOD

END_FUNCTION_BLOCK

// ---- POUs/99 Utilities/FB_TimeStampProvider.TcPOU
FUNCTION_BLOCK FB_TimeStampProvider

VAR
	fbLocalSystemTime: FB_LocalSystemTime;
END_VAR

fbLocalSystemTime();

METHOD FB_init : BOOL
VAR_INPUT
	bInitRetains : BOOL; // if TRUE, the retain variables are initialized (warm start / cold start)
	bInCopyCode : BOOL;  // if TRUE, the instance afterwards gets moved into the copy code (online change)
END_VAR
fbLocalSystemTime.bEnable := TRUE;		// A rising edge at this input triggers immediate synchronization of the internal time with the local Windows system time
fbLocalSystemTime.sNetID := '';  		// A string containing the network address of the TwinCAT computer whose time is to be used for the synchronization can be given here (type: T_AmsNetID). If it is to be run on the local computer, an empty string can be entered.
fbLocalSystemTime.dwCycle := 5; 				// Cycle time (in seconds) during which the function block resynchronizes its own time. Cyclic synchronization is activated after the first rising edge at the bEnable input. Default: Synchronization every 5 seconds.
fbLocalSystemTime.dwOpt := 1;							// Additional option parameters. The following parameters are currently available: Bit 0: If this is set, the Windows system time is additionally synchronized cyclically with the hardware clock (RTC) (corresponds to the function NT_SetTimeToRTCTime). Default: Activated.
fbLocalSystemTime.tTimeout := DEFAULT_ADS_TIMEOUT;		// This option is irrelevant for a Windows CE system.
END_METHOD

METHOD getTime : TIMESTRUCT

VAR_OUTPUT
	SystemTime : TIMESTRUCT;
END_VAR
getTime := fbLocalSystemTime.systemTime;
END_METHOD

END_FUNCTION_BLOCK

// ---- POUs/99 Utilities/_ss/FB_ModbusManager_1.TcPOU
FUNCTION_BLOCK FB_ModbusManager_1

VAR
	fbModbusMaster: FB_ModbusMaster_R2;
	
	
	
	aRequests_Read: 			ARRAY[0..(GVL.Max_Modbus_Requests_Read - 1)] OF POINTER TO ST_Modbus_ReadRequest;
	nIterator_Read_Insert: 		INT := 0;
	nIterator_Read_Action: 		INT := 0;
	nTotalRequests_Read: 		INT := 0;
	
	aRequests_Write: 			ARRAY[0..(GVL.Max_Modbus_Requests_Write - 1)] OF POINTER TO ST_Modbus_WriteRequest;
	nIterator_Write_Insert: 	INT := 0;
	nIterator_Write_Action:		INT := 0;
	nTotalRequests_Write: 		INT := 0;
	
	nNumRetries: 				INT := 0;
	bRead_or_Write_0_1:			BOOL := FALSE;
	bRequestAccepted: 			BOOL := FALSE;
	
	eSMState: (WAIT, REQUEST_READ, READING, READ, REQUEST_WRITE, WRITING, WRITTEN, REQUEST_READ_PRIORITY, READING_PRIORITY, READ_PRIORITY, REQUEST_WRITE_PRIORITY, WRITING_PRIORITY, WRITTEN_PRIORITY,ERROR) := WAIT;
	
	fbTON_RequestTimeout: TON := (PT := GVL.ModbusTimeout);
	tDelayBetweenMsg:	TIME := T#100MS;	
	fbTON_DelayBetweenMSG: TON := (PT := tDelayBetweenMsg, IN := FALSE);
	
	
	// These two buffers are for priority messages and will be serviced before requests in the other buffers (similar to QoS)
	aRequests_Read_Priority: 			ARRAY[0..(GVL.Max_Modbus_Requests_Read_Priority - 1)] OF POINTER TO ST_Modbus_ReadRequest;
	nIterator_Read_Insert_Priority: 	INT := 0;
	nIterator_Read_Action_Priority: 	INT := 0;
	nTotalRequests_Read_Priority: 		INT := 0;
	
	aRequests_Write_Priority: 			ARRAY[0..(GVL.Max_Modbus_Requests_Write_Priority - 1)] OF POINTER TO ST_Modbus_WriteRequest;
	nIterator_Write_Insert_Priority: 	INT := 0;
	nIterator_Write_Action_Priority:	INT := 0;
	nTotalRequests_Write_Priority: 		INT := 0;
	
	bRead_or_Write_0_1_Priority:		BOOL := FALSE;
	
END_VAR

fbModbusMaster();
fbTON_RequestTimeout(PT := GVL.ModbusTimeout);


CASE eSMState OF
	
	WAIT:
		// Wait for a message to be received in either the Rx or Tx buffers
		nNumRetries := 0;
		fbTON_DelayBetweenMSG(PT := tDelayBetweenMsg, IN := TRUE);
		
		IF fbTON_DelayBetweenMSG.Q THEN
			// Service priority writes first
			IF nTotalRequests_Write_Priority > 0 THEN
				eSMState := REQUEST_WRITE_PRIORITY;
			// Service priority reads second
			ELSIF nTotalRequests_Read_Priority > 0 THEN
				eSMState := REQUEST_READ_PRIORITY;
			// Else toggle betwweenm read and write
			ELSIF bRead_or_Write_0_1 THEN   // If there are no priority messages then serve the non-critical requests
				bRead_or_Write_0_1 := FALSE;
				IF nTotalRequests_Write > 0 THEN
					eSMState := REQUEST_WRITE;
				END_IF
			ELSE 
				bRead_or_Write_0_1 := TRUE;
				IF nTotalRequests_Read > 0 THEN
					eSMState := REQUEST_READ;	
				END_IF
			END_IF
			fbTON_DelayBetweenMSG.IN := FALSE;
		END_IF
		

		
	REQUEST_READ:
		fbModbusMaster.readRegs(ReadRequest := aRequests_Read[nIterator_Read_Action], bRequestAccepted => bRequestAccepted);
		IF bRequestAccepted THEN
			eSMState := READING;
			bRequestAccepted := FALSE;
			fbTON_RequestTimeout.IN := TRUE;
		END_IF
		// Send a read request to the modbus master, progress to READING if modbus master accepts
		
	READING:
	
		IF aRequests_Read[nIterator_Read_Action]^.bRequestCompleted = TRUE THEN
			eSMState := READ;
			fbTON_RequestTimeout.IN := FALSE;
		END_IF
		
		IF fbTON_RequestTimeout.Q THEN
			eSMState := REQUEST_READ; 
			nNumRetries := nNumRetries + 1;
			IF nNumRetries > GVL.ModbusMaxRetires THEN
				// ADD CODE HERE - Raise an error - and proceed to the next request - attach info about the request to the error so we can troubleshoot it
				eSMState := READ;
			END_IF
		END_IF
		
		// Stay in this state until the boolean pointer of job completed is set to true
		// Monitor the timeout timer and retry request if necessary
		
	READ:
		// Set the position in the ring buffer to 0 and iterate to the next, return to wait where the decision will be made to read or write
		aRequests_Read[nIterator_Read_Action] := 0;
		nIterator_Read_Action := nIterator_Read_Action + 1;
		
		IF nIterator_Read_Action > (GVL.Max_Modbus_Requests_Read - 1) THEN // return to 0 index if we are at the end of the buffer
			nIterator_Read_Action := 0;
		END_IF
		nTotalRequests_Read := nTotalRequests_Read - 1;
		eSMState := WAIT;
	
		
	REQUEST_WRITE:
		// Send a read request to the modbus master, progress to WRITING if modbus master accepts
		fbModbusMaster.writeRegs(WriteRequest := aRequests_Write[nIterator_Write_Action], bRequestAccepted => bRequestAccepted);
		IF bRequestAccepted THEN
			eSMState := WRITING;
			bRequestAccepted := FALSE;
			fbTON_RequestTimeout.IN := TRUE;
		END_IF
		
	WRITING:
		// Stay in this state until the boolean pointer of job completed is set to true
		IF aRequests_Write[nIterator_Write_Action]^.bRequestCompleted = TRUE THEN
			eSMState := WRITTEN;
			fbTON_RequestTimeout.IN := FALSE;
		END_IF
		
		IF fbTON_RequestTimeout.Q THEN
			eSMState := REQUEST_WRITE; 
			nNumRetries := nNumRetries + 1;
			IF nNumRetries > GVL.ModbusMaxRetires THEN
				// ADD CODE HERE - Raise an error - and proceed to the next request - attach info about the request to the error so we can troubleshoot it
				eSMState := WRITTEN;
			END_IF
		END_IF
		
		
	WRITTEN:
		// Set the position in the ring buffer to 0 and iterate to the next, return to wait where the decision will be made to read or write
		aRequests_Write[nIterator_Write_Action] := 0;
		nIterator_Write_Action := nIterator_Write_Action + 1;
		
		IF nIterator_Write_Action > (GVL.Max_Modbus_Requests_Write - 1) THEN
			nIterator_Write_Action := 0;
		END_IF
		
		nTotalRequests_Write := nTotalRequests_Write - 1;
		eSMState := WAIT;
		
		
	REQUEST_READ_PRIORITY:
		fbModbusMaster.readRegs(ReadRequest := aRequests_Read_Priority[nIterator_Read_Action_Priority], bRequestAccepted => bRequestAccepted);
		IF bRequestAccepted THEN
			eSMState := READING_PRIORITY;
			bRequestAccepted := FALSE;
			fbTON_RequestTimeout.IN := TRUE;
		END_IF
		// Send a read request to the modbus master, progress to READING if modbus master accepts
		
	READING_PRIORITY:
	
		IF aRequests_Read_Priority[nIterator_Read_Action_Priority]^.bRequestCompleted = TRUE THEN
			eSMState := READ_PRIORITY;
			fbTON_RequestTimeout.IN := FALSE;
		END_IF
		
		IF fbTON_RequestTimeout.Q THEN
			eSMState := REQUEST_READ_PRIORITY; 
			nNumRetries := nNumRetries + 1;
			IF nNumRetries > GVL.ModbusMaxRetires THEN
				// ADD CODE HERE - Raise an error - and proceed to the next request - attach info about the request to the error so we can troubleshoot it
				eSMState := READ_PRIORITY;
			END_IF
		END_IF
		
		// Stay in this state until the boolean pointer of job completed is set to true
		// Monitor the timeout timer and retry request if necessary
		
	READ_PRIORITY:
		// Set the position in the ring buffer to 0 and iterate to the next, return to wait where the decision will be made to read or write
		aRequests_Read_Priority[nIterator_Read_Action_Priority] := 0;
		nIterator_Read_Action_Priority := nIterator_Read_Action_Priority + 1;
		
		IF nIterator_Read_Action_Priority > (GVL.Max_Modbus_Requests_Read_Priority - 1) THEN // return to 0 index if we are at the end of the buffer
			nIterator_Read_Action_Priority := 0;
		END_IF
		nTotalRequests_Read_Priority := nTotalRequests_Read_Priority - 1;
		eSMState := WAIT;
	
		
	REQUEST_WRITE_PRIORITY:
		// Send a read request to the modbus master, progress to WRITING if modbus master accepts
		fbModbusMaster.writeRegs(WriteRequest := aRequests_Write_Priority[nIterator_Write_Action_Priority], bRequestAccepted => bRequestAccepted);
		IF bRequestAccepted THEN
			eSMState := WRITING_PRIORITY;
			bRequestAccepted := FALSE;
			fbTON_RequestTimeout.IN := TRUE;
		END_IF
		
	WRITING_PRIORITY:
		// Stay in this state until the boolean pointer of job completed is set to true
		IF aRequests_Write_Priority[nIterator_Write_Action_Priority]^.bRequestCompleted = TRUE THEN
			eSMState := WRITTEN_PRIORITY;
			fbTON_RequestTimeout.IN := FALSE;
		END_IF
		
		IF fbTON_RequestTimeout.Q THEN
			eSMState := REQUEST_WRITE_PRIORITY; 
			nNumRetries := nNumRetries + 1;
			IF nNumRetries > GVL.ModbusMaxRetires THEN
				// ADD CODE HERE - Raise an error - and proceed to the next request - attach info about the request to the error so we can troubleshoot it
				eSMState := WRITTEN_PRIORITY;
			END_IF
		END_IF
		
		
	WRITTEN_PRIORITY:
		// Set the position in the ring buffer to 0 and iterate to the next, return to wait where the decision will be made to read or write
		aRequests_Write_Priority[nIterator_Write_Action_Priority] := 0;
		nIterator_Write_Action_Priority := nIterator_Write_Action_Priority + 1;
		
		IF nIterator_Write_Action_Priority > (GVL.Max_Modbus_Requests_Write_Priority - 1) THEN
			nIterator_Write_Action_Priority := 0;
		END_IF
		
		nTotalRequests_Write_Priority := nTotalRequests_Write_Priority - 1;
		eSMState := WAIT;
		
	ERROR:
		//
		
END_CASE

METHOD addRequest_Read : BOOL
VAR_INPUT
	ReadRequest: POINTER TO ST_Modbus_ReadRequest;
END_VAR
IF aRequests_Read[nIterator_Read_Insert] = 0 THEN
	
	aRequests_Read[nIterator_Read_Insert] := ReadRequest;
	aRequests_Read[nIterator_Read_Insert]^.bRequestAccepted := FALSE;
	aRequests_Read[nIterator_Read_Insert]^.bRequestCompleted := FALSE;
	nIterator_Read_Insert := nIterator_Read_Insert + 1;
	
	IF nIterator_Read_Insert > (GVL.Max_Modbus_Requests_Read -1) THEN
		nIterator_Read_Insert := 0;
	END_IF
	
	nTotalRequests_Read := nTotalRequests_Read + 1;
	
	
	addRequest_Read := TRUE;
ELSE
	addRequest_Read := FALSE;	// A buffer overflow has occured here, add some error raising code here
END_IF
END_METHOD

METHOD addRequest_Read_Priority : BOOL
VAR_INPUT
	ReadRequest: POINTER TO ST_Modbus_ReadRequest;
END_VAR
IF aRequests_Read_Priority[nIterator_Read_Insert_Priority] = 0 THEN
	
	aRequests_Read_Priority[nIterator_Read_Insert_Priority] := ReadRequest;
	aRequests_Read_Priority[nIterator_Read_Insert_Priority]^.bRequestAccepted := FALSE;
	aRequests_Read_Priority[nIterator_Read_Insert_Priority]^.bRequestCompleted := FALSE;
	nIterator_Read_Insert_Priority := nIterator_Read_Insert_Priority + 1;
	
	IF nIterator_Read_Insert_Priority > (GVL.Max_Modbus_Requests_Read_Priority -1) THEN
		nIterator_Read_Insert_Priority := 0;
	END_IF
	
	nTotalRequests_Read_Priority := nTotalRequests_Read_Priority + 1;
	
	
	addRequest_Read_Priority := TRUE;
ELSE
	addRequest_Read_Priority := FALSE;	// A buffer overflow has occured here, add some error raising code here
END_IF
END_METHOD

METHOD addRequest_Write : BOOL
VAR_INPUT
	WriteRequest: POINTER TO ST_Modbus_WriteRequest;
END_VAR
IF aRequests_Write[nIterator_Write_Action] = 0 THEN
	aRequests_Write[nIterator_Write_Action] := WriteRequest;
	aRequests_Write[nIterator_Write_Action]^.bRequestAccepted := FALSE;
	aRequests_Write[nIterator_Write_Action]^.bRequestCompleted := FALSE;
	nIterator_Write_Insert := nIterator_Write_Insert + 1;
	
	IF nIterator_Write_Insert > (GVL.Max_Modbus_Requests_Write - 1) THEN
		nIterator_Write_Insert := 0;
	END_IF
	
	nTotalRequests_Write := nTotalRequests_Write + 1;
	
ELSE
	addRequest_Write := FALSE; // A buffer overflow has occured here, add some error raising code here
END_IF
END_METHOD

METHOD addRequest_Write_Priority : BOOL
VAR_INPUT
	WriteRequest: POINTER TO ST_Modbus_WriteRequest;
END_VAR
IF aRequests_Write_Priority[nIterator_Write_Insert_Priority] = 0 THEN
	
	aRequests_Write_Priority[nIterator_Write_Insert_Priority] := WriteRequest;
	aRequests_Write_Priority[nIterator_Write_Insert_Priority]^.bRequestAccepted := FALSE;
	aRequests_Write_Priority[nIterator_Write_Insert_Priority]^.bRequestCompleted := FALSE;
	nIterator_Write_Insert_Priority := nIterator_Write_Insert_Priority + 1;
	
	IF nIterator_Write_Insert_Priority > (GVL.Max_Modbus_Requests_Write_Priority - 1) THEN
		nIterator_Write_Insert_Priority := 0;
	END_IF
	
	nTotalRequests_Write_Priority := nTotalRequests_Write_Priority + 1;
	
ELSE
	addRequest_Write_Priority := FALSE; // A buffer overflow has occured here, add some error raising code here
END_IF
END_METHOD

METHOD FB_init : BOOL
VAR_INPUT
	bInitRetains : BOOL; // if TRUE, the retain variables are initialized (warm start / cold start)
	bInCopyCode : BOOL;  // if TRUE, the instance afterwards gets moved into the copy code (online change)
END_VAR

VAR
	i: INT := 0;
END_VAR
WHILE i < GVL.Max_Modbus_Requests_Read DO
	aRequests_Read[i] := 0;
	i := i + 1;
END_WHILE

i := 0;

WHILE i < GVL.Max_Modbus_Requests_Write DO
	aRequests_Write[i] := 0;
	i := i + 1;
END_WHILE
END_METHOD

END_FUNCTION_BLOCK

// ---- POUs/99 Utilities/_ss/FB_ModbusMaster_R2_1.TcPOU
FUNCTION_BLOCK FB_ModbusMaster_R2_1

VAR
	MB: ModbusRtuMaster_KL6x22B;
	
	nReadRegsVals: POINTER TO ARRAY[1..10] OF WORD;
	nWriteRegVals: ARRAY[1..10] OF WORD;
	
	
	bRequestFinshed : POINTER TO BOOL;
		
	nSlaveAddress : BYTE;
	nQtyWordsToRead : WORD;
	nQtyWordsToWrite : WORD;
	nAdrFirstSlaveRegisterRead : WORD;
	nAdrFirstSlaveRegisterWrite : WORD;
	nTimeout : TIME := T#5S;
	
	
	// State Machine
	eState: (IDLE, BUSY, ERROR) := IDLE;
	eSMState: (WAIT, READ_TRIG, READ, WRITE_TRIG, WRITE, ERROR) := WAIT;
	eSMState_prev:  (WAIT, READ_TRIG, READ, WRITE_TRIG, WRITE, ERROR) := WAIT;
	bBusy: BOOL;
	
	//eOperationType: (READ_OP, WRITE_OP, READWRITE_OP);
	eOperationType: E_AccessType;
	fbTrigger : R_TRIG;
	
	bOperationFirstRun: BOOL := TRUE;
	nNumRetries: INT := 0; 
	nRetryThreshold: INT := 10;

END_VAR

fbTrigger();

CASE eSMState OF
	WAIT :
		eState := IDLE;
		MB.ReadRegs(Execute := FALSE);
        MB.WriteRegs(Execute := FALSE);
		bBusy := FALSE;
		
		IF fbTrigger.Q THEN
			IF eOperationType = E_AccessType.WRITE THEN
				eSMState := WRITE_TRIG;
			ELSIF eOperationType = E_AccessType.READ THEN
				eSMState := READ_TRIG;
			END_IF
		END_IF
		
		
		
	READ_TRIG : 
		eState := BUSY;
		IF bOperationFirstRun THEN
			nNumRetries := 0;
			bOperationFirstRun := FALSE;
		END_IF
	
		IF eOperationType = E_AccessType.READ THEN
			
			 MB.ReadRegs(
				UnitID:= nSlaveAddress, 
				Quantity:= nQtyWordsToRead, 
				MBAddr:= nAdrFirstSlaveRegisterRead, 
				cbLength:= nQtyWordsToRead * 2,//SIZEOF(nReadRegsVals), 
				pMemoryAddr:= ADR(nReadRegsVals), 
				Execute:= TRUE, 
				Timeout:= nTimeout );
			
			
			IF NOT MB.BUSY THEN 
				MB.ReadRegs(Execute := FALSE );
				bBusy := TRUE;
				IF MB.Error THEN 
					eSMState_prev := eSMState;
					eSMState := ERROR;           // handle errors 
				ELSE 
					eSMState := READ; // [...]               // keep going 
				END_IF
			END_IF
		END_IF
		
		IF nNumRetries > nRetryThreshold THEN
			eSMState := WAIT;
		END_IF
		
		
	READ :
	
		IF NOT MB.BUSY THEN
			eSMState := WAIT;
			bRequestFinshed^ := TRUE;
			bBusy := FALSE;
			fbTrigger.CLK := FALSE;
			bOperationFirstRun := TRUE;
		ELSIF MB.Error THEN
			eSMState_prev := eSMState;
			eSMState := ERROR;
		END_IF
	
	
	
	WRITE_TRIG :

		IF bOperationFirstRun THEN
			nNumRetries := 0;
			bOperationFirstRun := FALSE;
		END_IF
	(*
		MB.WriteRegs(
			UnitID:= nSlaveAddress, 
			Quantity:= nQtyWordsToWrite, 
			MBAddr:= nAdrFirstSlaveRegisterWrite, 
			cbLength:= nQtyWordsToWrite * 2, 
			pMemoryAddr:= ADR(nWriteRegVals), 
			Execute:= TRUE, 
			Timeout:= nTimeout); 
		*)	
		
		MB.UnitID:= nSlaveAddress;
		MB.Quantity:=1;
		MB.MBAddr:= nAdrFirstSlaveRegisterWrite;
		MB.cbLength:= nQtyWordsToWrite * 2;
		MB.pMemoryAddr:= ADR(nWriteRegVals);
		MB.Execute:= TRUE;
		MB.Timeout:= nTimeout;
		MB.WriteSingleRegister();
		
			
		IF NOT MB.BUSY THEN 
			//MB.WriteRegs(Execute := FALSE );
			MB.Execute := FALSE;
			bBusy := TRUE;
			IF MB.Error THEN 
				eSMState_prev := eSMState;
				eSMState := ERROR;           				// handle errors 
			ELSE 
				eSMState := WRITE;			            // keep going 
			END_IF
		END_IF

	
		
	WRITE:
		IF NOT MB.BUSY THEN
			eSMState := WAIT;
			bRequestFinshed^ := TRUE;
			bBusy := FALSE;
			fbTrigger.CLK := FALSE;
			bOperationFirstRun := TRUE;
		ELSIF MB.Error THEN
			eSMState_prev := eSMState;
			eSMState := ERROR;
		END_IF
	
		
	ERROR:
		nNumRetries := nNumRetries + 1;
		IF nNumRetries > nRetryThreshold THEN
			eState := ERROR;
			eSMState := WAIT;
		ELSE
			eSMState := eSMState_prev;
		END_IF
		 
			
		

END_CASE

METHOD Error : BOOL
VAR_INPUT
END_VAR
Error := MB.Error;
END_METHOD

METHOD FB_init : BOOL
VAR_INPUT
	bInitRetains : BOOL; // if TRUE, the retain variables are initialized (warm start / cold start)
	bInCopyCode : BOOL;  // if TRUE, the instance afterwards gets moved into the copy code (online change)
END_VAR
END_METHOD

METHOD isBusy : BOOL
isBusy := bBusy;
END_METHOD

METHOD readRegs : BOOL
VAR_INPUT
	ReadRequest: POINTER TO ST_Modbus_ReadRequest;
END_VAR

VAR_OUTPUT
	bRequestAccepted: BOOL;
END_VAR
IF eSMState = WAIT THEN
	eOperationType := E_AccessType.READ;
	nReadRegsVals := ADR(ReadRequest^.ReadRegsVals);
	nSlaveAddress := UINT_TO_BYTE(ReadRequest^.SlaveAddress);
	nQtyWordsToRead := UINT_TO_WORD(ReadRequest^.QtyWordsToRead);
	nAdrFirstSlaveRegisterRead := UINT_TO_WORD(ReadRequest^.AdrFirstSlaveRegisterRead);
	fbTrigger.CLK := TRUE;
	bRequestAccepted := TRUE;
	bBusy := TRUE;
	bRequestFinshed := ADR(ReadRequest^.bRequestCompleted);
	eSMState := READ_TRIG;
END_IF
END_METHOD

METHOD writeReg : BOOL
VAR_INPUT
	WriteRegVal: WORD;
	SlaveAddress : UINT;
	AdrFirstSlaveRegisterWrite : UINT;
	bRequestCompleted : POINTER TO BOOL;
	
	WriteRequest: ST_Modbus_WriteRequest;
END_VAR

VAR_OUTPUT
	bRequestAccepted: BOOL := FALSE;
END_VAR
(* IF eState = WAIT THEN
	eOperationType := E_AccessType.WRITE;
	//nWriteRegVals[0] := WriteRegVal;
	nWriteRegVals[1] := WriteRegVal;
	nWriteRegVals[1] := WriteRequest.
	nSlaveAddress := UINT_TO_BYTE(SlaveAddress);
	nQtyWordsToWrite := 1;
	nAdrFirstSlaveRegisterWrite := UINT_TO_BYTE(AdrFirstSlaveRegisterWrite);
	bRequestAccepted := TRUE;
	bRequestFinshed := bRequestCompleted;
	fbTrigger.CLK := TRUE;
	eState := WRITE_TRIG;
	
END_IF
*) 

// This needs to be re written to suit ST requests
END_METHOD

METHOD writeRegs : BOOL
VAR_INPUT

	
	WriteRequest: POINTER TO ST_Modbus_WriteRequest;

END_VAR

VAR_OUTPUT
	bRequestAccepted: BOOL := FALSE;
END_VAR
IF eSMState = WAIT THEN
	eOperationType := E_AccessType.WRITE;
	nWriteRegVals := WriteRequest^.WriteRegVals;
	nSlaveAddress := UINT_TO_BYTE(WriteRequest^.SlaveAddress);
	nQtyWordsToWrite := UINT_TO_WORD(WriteRequest^.QtyWordsToWrite);
	nAdrFirstSlaveRegisterWrite := UINT_TO_WORD(WriteRequest^.AdrFirstSlaveRegisterWrite);
	bRequestFinshed := ADR(WriteRequest^.bRequestCompleted);	
	fbTrigger.CLK := TRUE;
	bRequestAccepted := TRUE;
	
	eSMState := WRITE_TRIG;
END_IF
END_METHOD

END_FUNCTION_BLOCK

// ---- POUs/LFT/FB_ParameterCoE_ReadWrite_GenC.TcPOU
(*-----------------------------------------------------------------------------------------------------------
	Function: CoE/Sdo Acces for Read and Write Services on MOVI-C devices of SEW EURODRIVE
	Version: 1.4
	Date: 2022-07-01
	Author: Christian Bolz; SE-PAS
	
	Change-Log:
		2018-04-25: V1.1:
					- Functionality is working properly
					- first tests
		2022-07-15: V1.4
					- Changing Service Input to Enumeration
					- Chaning Axis Number Input to Enumeration
					- Inserting missing inputs as enumeration as output of the FB (eConfigurationState)
============================================================================================================*)	


FUNCTION_BLOCK FB_ParameterCoE_ReadWrite_GenC
VAR_INPUT
	xExecute						: BOOL;						//Execute FoE-Service
	amsEthercatMaster_NetID			: T_AmsNetId;				//EtherCAT Master Net-ID
	nEthercatSlave_Address			: UINT;						//EtherCAT Adress Slave
	eAxisNumber						: E_AxisNumberCoE;			//1-->Modular-SingleAxis/Modular-DoubleAxisLEFT/SystemAxis; 2-->Modular-DoubleAxisRIGHT
	eCoEService						: E_CoEService; 			//1-->Read / 2-->write
	nIndex							: UINT;						//Parameterindex of EtherCAT Slave
	nSubIndex 						: BYTE;						//Subindex of Parameter
	nWriteValue						: DINT;						//Value to write to EtherCAT Slave
	nByteSize						: UINT;

END_VAR
VAR_OUTPUT
	xError_CoE						: BOOL;						//TRUE-->Error during CoE-service
	xCoEDone						: BOOL;						//TRUE-->CoE-access successful
	nErrId_ADS						: UDINT;					//ADS Error-ID of FoE-service
	xCoEBusy						: BOOL;						//TRUE-->Function block busy
	eActualCoEService				: E_COEService;				//Selected CoE-service
	xInit							: BOOL;						//TRUE-->parametrization OK / FALSE--> parmetrization not OK
	nReadValue						: DINT;						//Value that is read from EtherAT Slave
	eConfigurationStateCoE			: E_ConfigurationStateCoE;
END_VAR
VAR
	(*------------------------------------------------------------------------------------------------------
		READ/WRITE Function Blocks
	=======================================================================================================*)
	fbFB_EcCoeSdoReadEx: FB_EcCoeSdoReadEx;
	fbFB_EcCoeSdoWriteEx: FB_EcCoeSdoWriteEx;

	(*------------------------------------------------------------------------------------------------------
		BUFFER
	=======================================================================================================*)
	buffer_read_0						: BYTE;
	buffer_write_0						: BYTE;
	buffer_read_1						: BYTE;					//Buffer where the read value is stored, ParamSize := BYTE
	buffer_write_1						: BYTE;					//Buffer where the value to write is stored, ParamSize := BYTE
	buffer_read_2						: INT;					//Buffer where the read value is stored, ParamSize := INT
	buffer_write_2						: INT;					//Buffer where the value to write is stored, ParamSize := INT
	buffer_read_4						: DINT;					//Buffer where the read value is stored, ParamSize := DINT
	buffer_write_4						: DINT;					//Buffer where the value to write is stored, ParamSize := DINT
	(*------------------------------------------------------------------------------------------------------
		GENERAL VARS
	=======================================================================================================*)	
	iState_CoEWrite					: INT;					//state of FoE write service
	iState_CoERead					: INT;					//state of FoE read service
END_VAR

IF xExecute THEN
	IF NOT xInit THEN
		xError_CoE := FALSE;
		xCoEDone := FALSE;
		
		IF amsEthercatMaster_NetID<>'' AND nEthercatSlave_Address<>0  AND nByteSize<>0 AND nByteSize<=4 AND nByteSize<>3 THEN
			xInit := TRUE;
			eConfigurationStateCoE := 0;
		ELSE
			IF amsEthercatMaster_NetID='' THEN
				eConfigurationStateCoE := 1;
			END_IF
			IF nEthercatSlave_Address=0 THEN
				eConfigurationStateCoE := 2;
			END_IF
			IF nByteSize=0 OR nByteSize>4 OR nByteSize=3 OR nByteSize = 1 THEN
				eConfigurationStateCoE := 3;
			END_IF
		END_IF		
	END_IF
	
	CASE eCoEService OF
		0:
			eActualCoEService := 0;
		1:
		
			CASE eAxisNumber OF
				1:;
				2:
					nIndex := nIndex+16#1000;
			END_CASE
			
			IF xInit THEN
				ACT_Read();	
			END_IF
			
		2:
			CASE eAxisNumber OF
				1:;
				2:
					nIndex := nIndex+16#1000;
			END_CASE
			
			IF xInit THEN
				ACT_Write();
			end_if
	END_CASE
	
ELSE
	xInit := FALSE;
	xCoEBusy := FALSE;
	xError_CoE := FALSE;
	
	nReadValue := 0;
	iState_CoEWrite := 0;
	iState_CoERead := 0;
	xCoEDone := FALSE;
	nErrId_ADS := 0;
	fbFB_EcCoeSdoReadEx(pDstBuf := ADR(buffer_read_0),
						cbBufLen := SIZEOF(buffer_read_0));
END_IF

IF NOT xExecute  AND NOT xCoEBusy THEN
	xError_CoE := FALSE;
	xInit := FALSE;
	nErrId_ADS := 0;
ELSIF xError_CoE AND xCoEBusy AND NOT xExecute THEN
	xError_CoE := FALSE;
	iState_CoEWrite := 0;
	iState_CoERead := 0;
	xInit := FALSE;
	
END_IF

ACTION ACT_Read:
eActualCoEService := 1;
CASE iState_CoERead OF
	0:
		fbFB_EcCoeSdoReadEx(bExecute := FALSE,
			sNetId := amsEthercatMaster_NetID,
			nSlaveAddr := nEthercatSlave_Address,
			nSubINdex := nSubIndex,
			nIndex := nIndex,
			(*pDstBuf := ADR(buffer_read),
			cbBufLen := 4(*SIZEOF(buffer_read)*),*)
			tTimeout := T#200MS,
			bBusy => xCoEBusy,
			bError => xError_CoE,
			nErrId => nErrId_ADS,
			bCompleteAccess := FALSE);
			
			CASE nByteSize OF
				1:
					fbFB_EcCoeSdoReadEx(pDstBuf := ADR(buffer_read_1),
						cbBufLen := SIZEOF(buffer_read_1));
				2:
					fbFB_EcCoeSdoReadEx(pDstBuf := ADR(buffer_read_2),
						cbBufLen := SIZEOF(buffer_read_2));
				4:
					fbFB_EcCoeSdoReadEx(pDstBuf := ADR(buffer_read_4),
						cbBufLen := SIZEOF(buffer_read_4));
			END_CASE
			
			iState_CoERead := iState_CoERead+1;
		1:
			fbFB_EcCoeSdoReadEx(bExecute := TRUE);
			
			IF NOT fbFB_EcCoeSdoReadEx.bBusy THEN
				IF fbFB_EcCoeSdoReadEx.bError THEN
					iState_CoERead := 101;
					nErrId_ADS := fbFB_EcCoeSdoReadEx.nErrId;
				ELSE
					CASE nByteSize OF
						1:
							nReadValue := BYTE_TO_DINT(buffer_read_1);
						2:
							nReadValue := INT_TO_DINT(buffer_read_2);
						4:
							nReadValue := buffer_read_4;
					END_CASE
					
					iState_CoERead := 1000;
				END_IF
			END_IF
		
		101:
			xError_CoE := TRUE;
		1000:
			xCoEDone := TRUE;
			nErrId_ADS := 0;
			xError_CoE := FALSE;
END_CASE
END_ACTION

ACTION ACT_Write:
eActualCoEService := 2;
CASE iState_CoEWrite OF
	0:
		CASE nByteSize OF 
			1:
				buffer_write_1 := DINT_TO_BYTE(nWriteValue);
			2:
				buffer_write_2 := DINT_TO_INT(nWriteValue);
			4:
				buffer_write_4 := nWriteValue;
		END_CASE
		
		
		iState_CoEWrite := iState_CoEWrite+1;
	1:
		fbFB_EcCoeSdoWriteEx(bExecute := FALSE,
			sNetId := amsEthercatMaster_NetID,
			nSlaveAddr := nEthercatSlave_Address,
			nSubINdex := nSubIndex,
			nIndex := nIndex,
			tTimeout := T#200MS,
			bBusy => xCoEBusy,
			bError => xError_CoE,
			nErrId => nErrId_ADS,
			bCompleteAccess := FALSE);
			
			CASE nByteSize OF
				1:
					fbFB_EcCoeSdoWriteEx(pSrcBuf := ADR(buffer_write_1),
						cbBufLen := SIZEOF(buffer_write_1));
				2:
					fbFB_EcCoeSdoWriteEx(pSrcBuf := ADR(buffer_write_2),
						cbBufLen := SIZEOF(buffer_write_2));
				4:
					fbFB_EcCoeSdoWriteEx(pSrcBuf := ADR(buffer_write_4),
						cbBufLen := SIZEOF(buffer_write_4));
			END_CASE
			
			iState_CoEWrite := iState_CoEWrite+1;
		2:
			fbFB_EcCoeSdoWriteEx(bExecute := TRUE);
			
			IF NOT fbFB_EcCoeSdoWriteEx.bBusy THEN
				IF fbFB_EcCoeSdoWriteEx.bError THEN
					iState_CoEWrite := 202;
					nErrId_ADS := fbFB_EcCoeSdoWriteEx.nErrId;
				ELSE
					
					iState_CoEWrite := 1000;
				END_IF
			END_IF
		
		202:
			xError_CoE := TRUE;
		1000:
			xCoEDone := TRUE;
			nErrId_ADS := 0;
			xError_CoE := FALSE;
END_CASE
END_ACTION

END_FUNCTION_BLOCK

// ---- POUs/POP/FB_ActuatorLinear.TcPOU
FUNCTION_BLOCK FB_ActuatorLinear 

VAR	
	axis: 				AXIS_REF;
	power: 				MC_Power;
	powerOutputs: 		ST_McOutputs;
	moveAbs: 			MC_MoveAbsolute;
	moveAbsOutputs: 	ST_McOutputs;
	reset: 				MC_Reset;
	resetOut: 			ST_McOutputs;
	home:				MC_Home;
	
	
	sID: STRING;
	sDescr: STRING;
	
	
	nLead: UINT := 5;  			// mm per 360deg  - NOT EFFECTIVE YET BECAUSE PITCH IS CURRENTLY HANDLED IN THE AXIS CONFIG
	nStroke: UINT := 100;  		// length of travel
	nHomeOffset: UINT := 0; 	// offset distance from hard-stop for home
	nMaxVel: UINT := 300; 		// mm/s
	nPercentMove: LREAL := 100; 	// % of the full extent of movement (starting from position 0)
	
	eSMState: (INIT, ENABLE, WAIT, FWD_TRIG, FWD, REV_TRIG, REV, ERROR, RESET, HOMING, HOME) := INIT;
	
	fbTONDelay: TON := (PT := T#5S);
	bFirstRun: BOOL := TRUE;
	

	
END_VAR

ActMove();
ActPower();
ActReset();
fbTONDelay();


CASE eSMState OF
	
	INIT:

		IF bFirstRun THEN
			fbTONDelay.IN := TRUE;
			bFirstRun := FALSE;
		END_IF
		
		moveAbs.Execute := FALSE;
		moveAbs.Execute := FALSE;
		reset.Execute := FALSE;
		
		
		IF fbTONDelay.Q THEN
			eSMState := ENABLE;
			fbTONDelay.IN := FALSE;	
			bFirstRun := TRUE;
		END_IF
		
		
		
		
	ENABLE:
	
		IF bFirstRun THEN
			fbTONDelay.IN := TRUE;
			bFirstRun := FALSE;
		END_IF
	
		
		power.Enable := TRUE;
		power.Enable_Positive := TRUE;
		power.Enable_Negative := TRUE;
		
		
		IF power.Status THEN
			eSMState := WAIT;
			fbTONDelay.IN := FALSE;	
			bFirstRun := TRUE;
		(* ELSIF power.Error AND fbTONDelay.Q THEN
			eSMState := ERROR;
			fbTONDelay.IN := FALSE;
			bFirstRun := TRUE; *)
		END_IF
		
	WAIT:
		// Handle eStateTarget command requests here 
		//IF eStateTarget := E_DeviceState.
		
	
	HOMING:
		
		
	FWD_TRIG:
			
			moveAbs.Position := - nStroke * (nPercentMove / 100);		(* mm *)
			moveAbs.Velocity := nMaxVel/2;		(* mm/s *)
			moveAbs.BufferMode := MC_Buffered;  
			moveAbs.Execute := TRUE;
			
			IF moveAbs.Active THEN
				moveAbs.Execute := FALSE;
				fbTONDelay.IN := FALSE;
				eSMState := FWD;
				bFirstRun := TRUE;
			ELSIF moveAbs.CommandAborted OR moveAbs.Error THEN
				eSMState := ERROR;
				bFirstRun := TRUE;
				moveAbs.Execute := FALSE;
			END_IF
				
	FWD:
			eSMState := INIT;
			//eState := FWD;
			
			
			
			
	REV_TRIG:
	
			moveAbs.Position := - (0 + nHomeOffset)  * (nPercentMove / 100);		(* mm *)
			moveAbs.Velocity := nMaxVel/2;										(* mm/s *)
			moveAbs.BufferMode := MC_Buffered;  
			moveAbs.Execute := TRUE;
			
			IF moveAbs.Active THEN
				moveAbs.Execute := FALSE;
				fbTONDelay.IN := FALSE;
				eSMState := REV;
				bFirstRun := TRUE;
			ELSIF moveAbs.CommandAborted OR moveAbs.Error THEN
				eSMState := ERROR;
				bFirstRun := TRUE;
				moveAbs.Execute := FALSE;
			END_IF
			
	REV:
			eSMState := INIT;
			

	ERROR:
			IF axis.Status.Error THEN
				eSMState := RESET;	(* axis error requires reset *)
			ELSE
				eSMState := INIT;		(* function block errors don't need a reset *)
			END_IF
	
	RESET:
	
			IF bFirstRun THEN
				fbTONDelay.IN := TRUE;
				bFirstRun := FALSE;
			END_IF
		
			reset.Execute := TRUE;
			
			IF reset.Done AND fbTONDelay.Q THEN
				eSMState := INIT;
				fbTONDelay.IN := FALSE;
				bFirstRun := TRUE;
			ELSIF reset.Error AND fbTONDelay.Q THEN
				eSMState := ERROR; // the example code pointed this to reset
				fbTONDelay.IN := FALSE;
				bFirstRun := TRUE;
			END_IF
	
	
END_CASE

ACTION ActMove:
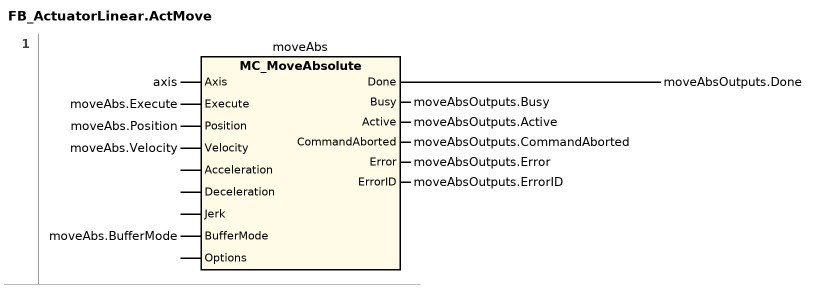
// NETWORK 1
moveAbs(
    Axis := axis,
    Execute := moveAbs.Execute,
    Position := moveAbs.Position,
    Velocity := moveAbs.Velocity,
    BufferMode := moveAbs.BufferMode,
    Busy => moveAbsOutputs.Busy,
    Active => moveAbsOutputs.Active,
    CommandAborted => moveAbsOutputs.CommandAborted,
    Error => moveAbsOutputs.Error,
    ErrorID => moveAbsOutputs.ErrorID); // MC_MoveAbsolute
moveAbsOutputs.Done := moveAbs.Done;
END_ACTION

ACTION ActMove_1:
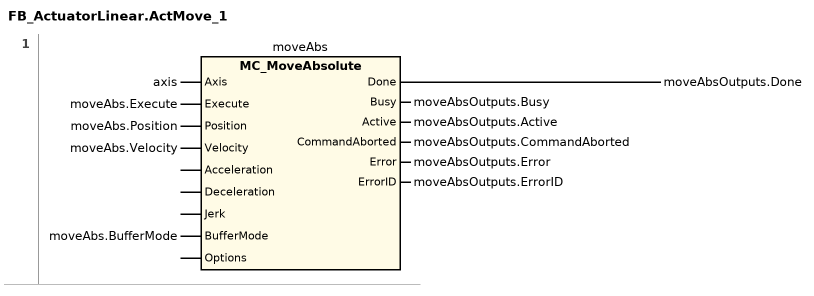
// NETWORK 1
moveAbs(
    Axis := axis,
    Execute := moveAbs.Execute,
    Position := moveAbs.Position,
    Velocity := moveAbs.Velocity,
    BufferMode := moveAbs.BufferMode,
    Busy => moveAbsOutputs.Busy,
    Active => moveAbsOutputs.Active,
    CommandAborted => moveAbsOutputs.CommandAborted,
    Error => moveAbsOutputs.Error,
    ErrorID => moveAbsOutputs.ErrorID); // MC_MoveAbsolute
moveAbsOutputs.Done := moveAbs.Done;
END_ACTION

ACTION ActPower:
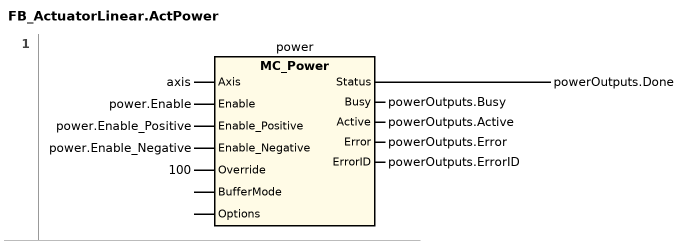
// NETWORK 1
power(
    Axis := axis,
    Enable := power.Enable,
    Enable_Positive := power.Enable_Positive,
    Enable_Negative := power.Enable_Negative,
    Override := 100,
    Busy => powerOutputs.Busy,
    Active => powerOutputs.Active,
    Error => powerOutputs.Error,
    ErrorID => powerOutputs.ErrorID); // MC_Power
powerOutputs.Done := power.Status;
END_ACTION

ACTION ActReset:
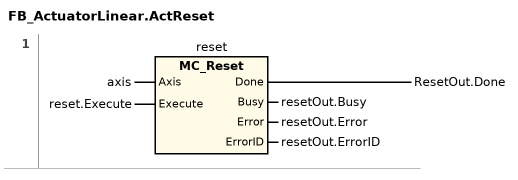
// NETWORK 1
reset(
    Axis := axis,
    Execute := reset.Execute,
    Busy => resetOut.Busy,
    Error => resetOut.Error,
    ErrorID => resetOut.ErrorID); // MC_Reset
ResetOut.Done := reset.Done;
END_ACTION

METHOD extend : BOOL
VAR_INPUT
END_VAR
IF eSMState = WAIT THEN
	eSMState := FWD_TRIG;
	nPercentMove := 100;
	extend := TRUE;
ELSE
	extend := FALSE;
END_IF
END_METHOD

METHOD FB_init : BOOL
VAR_INPUT
	bInitRetains : BOOL; // if TRUE, the retain variables are initialized (warm start / cold start)
	bInCopyCode : BOOL;  // if TRUE, the instance afterwards gets moved into the copy code (online change)
	
	ID: STRING;
	Descr: STRING;
	
	Lead: UINT;  			// mm per 360deg
	Stroke: UINT;  		// length of travel
	HomeOffset: UINT; 	// offset distance from hard-stop for home
END_VAR

sID := ID;
sDescr := Descr;

nLead := Lead;
nStroke := Stroke;
nHomeOffset := HomeOffset;
END_METHOD

METHOD initialise : BOOL
VAR_INPUT
	
	Lead: UINT;  			// mm per 360deg
	Stroke: UINT;  		// length of travel
	HomeOffset: UINT; 	// offset distance from hard-stop for home
END_VAR
nLead := Lead;
nStroke := Stroke;
nHomeOffset := HomeOffset;
END_METHOD

METHOD moveToPos : BOOL
VAR_INPUT
	PercStroke: LREAL;
END_VAR
IF eSMState = WAIT THEN
	eSMState := FWD_TRIG;
	nPercentMove := PercStroke;
	moveToPos := TRUE;
ELSE
	moveToPos := FALSE;
END_IF
END_METHOD

METHOD retract : BOOL
VAR_INPUT
END_VAR
IF eSMState = WAIT THEN
	eSMState := REV_TRIG;
	nPercentMove := 100;
	retract := TRUE;
ELSE
	retract := FALSE;
END_IF
END_METHOD

END_FUNCTION_BLOCK

// ---- POUs/POP/FB_BaseMotor.TcPOU
FUNCTION_BLOCK FB_BaseMotor

VAR
	mcAxis: 			AXIS_REF;
	eSMState:			E_MoveState;
	
	mcPower: 			MC_Power;
	mcPower_Outputs:	ST_McOutputs;
	
	mcReset: 			MC_Reset;
	mcReset_Outputs:	ST_McOutputs;
	
	mcStop:				MC_Stop;
	mcStop_Outputs:		ST_McOutputs;
	
	mcMoveAbs1: 			MC_MoveAbsolute;
	mcMoveAbs1_Outputs: 	ST_McOutputs;

	mcMoveAbs2: 			MC_MoveAbsolute;
	mcMoveAbs2_Outputs: 	ST_McOutputs;
	
	mcHome:				MC_Home;
	mcHome_Outputs:		ST_McOutputs;
	
END_VAR

(* update the axis status at the beginning of each cycle *)
mcAxis();

(* move axis using a state machine *)
CASE eSMState OF

	MOVESTATE_INIT :	(* initialisation *)
		(* initialize all function blocks *)
		mcMoveAbs1.Execute := FALSE;
		mcReset.Execute := FALSE;
		eSMState := MOVESTATE_ENABLE;

	MOVESTATE_ENABLE :
		mcPower.Enable := TRUE;
		mcPower.Enable_Positive := TRUE;
		mcPower.Enable_Negative := TRUE;
		IF mcPower.Status THEN
			eSMState := MOVESTATE_FORWARD;
		ELSIF mcPower.Error THEN
			eSMState := MOVESTATE_ERROR;
		END_IF

	MOVESTATE_FORWARD :							(* start to first position *)
		mcMoveAbs1.Position := 1500;				(* start to intermediate tartet position *)
		mcMoveAbs1.Velocity := 500;				(* medium velocity level *)
		mcMoveAbs1.BufferMode := MC_Buffered;
		mcMoveAbs1.Execute := TRUE;
		IF mcMoveAbs1.Active  THEN
			(* axis is executing job but is not yet finished *)
			mcMoveAbs1.Execute := FALSE;
			(* leave this state and buffer a second command *)
			eSMState := MOVESTATE_NEWTARGETPOSITION;
		ELSIF mcMoveAbs1.CommandAborted OR mcMoveAbs1.Error THEN
			eSMState := MOVESTATE_ERROR;
		END_IF

	MOVESTATE_NEWTARGETPOSITION :						(* change target position while moving *)
		(* start a buffered motion command while axis is moving *)
		mcMoveAbs2.Position := 5000;						(* start to final target *)
		mcMoveAbs2.Velocity := 1500;						(* increase velocity *)
		mcMoveAbs2.BufferMode := MC_BlendingPrevious; 		(* use velocity of previous command till intermediate target position position *)
		mcMoveAbs2.Execute := TRUE;
		IF mcMoveAbs2.Done THEN
			mcMoveAbs2.Execute := FALSE;
			eSMState := MOVESTATE_BACKWARDS;
		ELSIF mcMoveAbs2.CommandAborted OR mcMoveAbs2.Error THEN
			eSMState := MOVESTATE_ERROR;
		END_IF

	MOVESTATE_BACKWARDS :							(* move back to initial position *)
		mcMoveAbs1.Position := 100;					(* position close to initial position *)
		mcMoveAbs1.Velocity := 2000;				(* high velocity *)
		mcMoveAbs1.BufferMode := MC_Buffered;
		mcMoveAbs1.Execute := TRUE;
		IF mcMoveAbs1.Active THEN
			(* axis is executing job but is not yet finished *)
			mcMoveAbs1.Execute := FALSE;
			(* leave this state and buffer a second command *)
			eSMState := MOVESTATE_BACKWARDSSLOW;
		ELSIF mcMoveAbs1.CommandAborted OR mcMoveAbs1.Error THEN
			eSMState := MOVESTATE_ERROR;
		END_IF

	MOVESTATE_BACKWARDSSLOW :						(* move back to initial position *)
		(* start a buffered motion command while axis is moving *)
		mcMoveAbs2.Position := 0;					(* back to initial position *)
		mcMoveAbs2.Velocity := 100; 				(* slow velocity *)
		mcMoveAbs2.BufferMode := MC_BlendingNext; 	(* use velocity from first target position *)
		mcMoveAbs2.Execute := TRUE;
		IF mcMoveAbs2.Done THEN
			mcMoveAbs2.Execute := FALSE;
			eSMState := MOVESTATE_FORWARD;
		ELSIF mcMoveAbs2.CommandAborted OR mcMoveAbs2.Error THEN
			eSMState := MOVESTATE_ERROR;
		END_IF

	MOVESTATE_ERROR :
		IF mcAxis.Status.Error THEN
			eSMState := MOVESTATE_RESET;			(* axis error requires reset *)
		ELSE
			eSMState := MOVESTATE_INIT;			(* function block errors don't need a reset *)
		END_IF

	MOVESTATE_RESET :
		mcReset.Execute := TRUE;
		IF mcReset.Done THEN
			eSMState := MOVESTATE_INIT;
		ELSIF mcReset.Error THEN
			eSMState := MOVESTATE_INIT; 			(* can't do anything here *)
		END_IF

END_CASE

mcPower(Axis := mcAxis, 
		Enable := mcPower.Enable, 
		Enable_Positive := mcPower.Enable_Positive, 
		Enable_Negative := mcPower.Enable_Negative, 
		Override := 100, 
		Status => mcPower_Outputs.Done, 
		Busy => mcPower_Outputs.Busy, 
		Active => mcPower_Outputs.Active, 
		Error => mcPower_Outputs.Error, 
		ErrorID => mcPower_Outputs.ErrorID);


mcMoveAbs1(Axis := mcAxis,
			Execute := mcMoveAbs1.Execute,
			Position := mcMoveAbs1.Position,
			Velocity := mcMoveAbs1.Velocity,
			BufferMode := mcMoveAbs1.BufferMode,
			Done => mcMoveAbs1_Outputs.Done,
			Busy => mcMoveAbs1_Outputs.Busy,
			Active => mcMoveAbs1_Outputs.Active,
			CommandAborted => mcMoveAbs1_Outputs.CommandAborted,
			Error => mcMoveAbs1_Outputs.Error,
			ErrorID => mcMoveAbs1_Outputs.ErrorID);
			
mcMoveAbs2(Axis := mcAxis,
			Execute := mcMoveAbs1.Execute,
			Position := mcMoveAbs1.Position,
			Velocity := mcMoveAbs1.Velocity,
			BufferMode := mcMoveAbs1.BufferMode,
			Done => mcMoveAbs1_Outputs.Done,
			Busy => mcMoveAbs1_Outputs.Busy,
			Active => mcMoveAbs1_Outputs.Active,
			CommandAborted => mcMoveAbs1_Outputs.CommandAborted,
			Error => mcMoveAbs1_Outputs.Error,
			ErrorID => mcMoveAbs1_Outputs.ErrorID);
			
			
mcReset(Axis := mcAxis,
		Execute := mcReset.Execute,
		Done => mcReset_Outputs.Done,
		Busy => mcReset_Outputs.Busy,
		Error => mcReset_Outputs.Error,
		ErrorID => mcReset_Outputs.ErrorID);
	
// ActPower();	(* call the power function block *)
//ActMove();	(* call the move function block *)
//ActReset();	(* call the reset function block *)

ACTION ActMove:
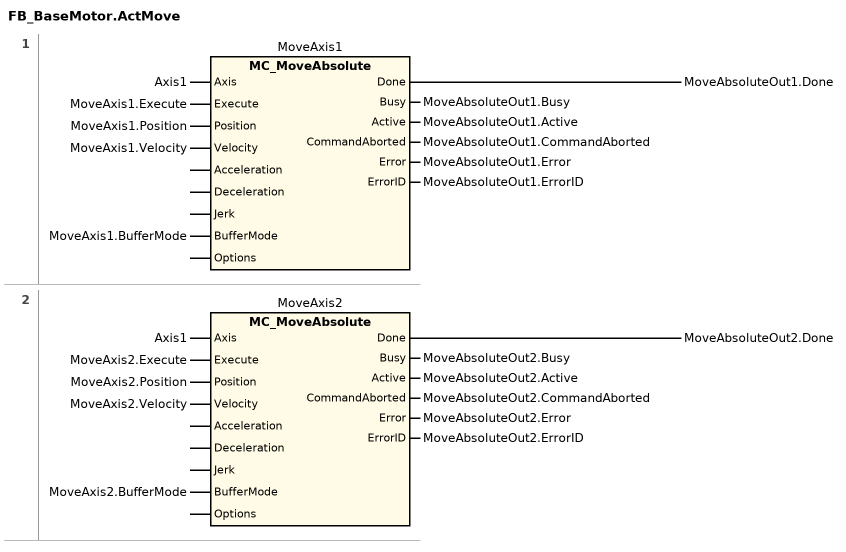
// NETWORK 1
MoveAxis1(
    Axis := Axis1,
    Execute := MoveAxis1.Execute,
    Position := MoveAxis1.Position,
    Velocity := MoveAxis1.Velocity,
    BufferMode := MoveAxis1.BufferMode,
    Busy => MoveAbsoluteOut1.Busy,
    Active => MoveAbsoluteOut1.Active,
    CommandAborted => MoveAbsoluteOut1.CommandAborted,
    Error => MoveAbsoluteOut1.Error,
    ErrorID => MoveAbsoluteOut1.ErrorID); // MC_MoveAbsolute
MoveAbsoluteOut1.Done := MoveAxis1.Done;

// NETWORK 2
MoveAxis2(
    Axis := Axis1,
    Execute := MoveAxis2.Execute,
    Position := MoveAxis2.Position,
    Velocity := MoveAxis2.Velocity,
    BufferMode := MoveAxis2.BufferMode,
    Busy => MoveAbsoluteOut2.Busy,
    Active => MoveAbsoluteOut2.Active,
    CommandAborted => MoveAbsoluteOut2.CommandAborted,
    Error => MoveAbsoluteOut2.Error,
    ErrorID => MoveAbsoluteOut2.ErrorID); // MC_MoveAbsolute
MoveAbsoluteOut2.Done := MoveAxis2.Done;
END_ACTION

ACTION ActPower:
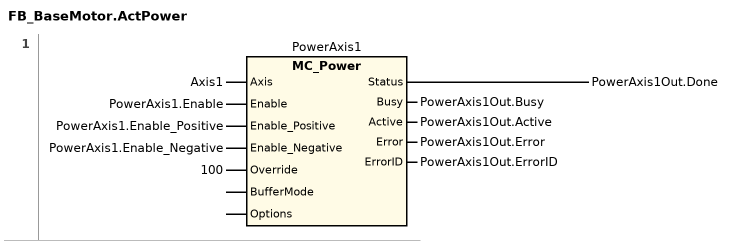
// NETWORK 1
PowerAxis1(
    Axis := Axis1,
    Enable := PowerAxis1.Enable,
    Enable_Positive := PowerAxis1.Enable_Positive,
    Enable_Negative := PowerAxis1.Enable_Negative,
    Override := 100,
    Busy => PowerAxis1Out.Busy,
    Active => PowerAxis1Out.Active,
    Error => PowerAxis1Out.Error,
    ErrorID => PowerAxis1Out.ErrorID); // MC_Power
PowerAxis1Out.Done := PowerAxis1.Status;
END_ACTION

ACTION ActReset:
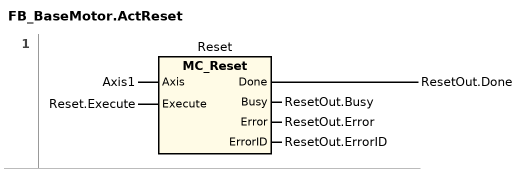
// NETWORK 1
Reset(
    Axis := Axis1,
    Execute := Reset.Execute,
    Busy => ResetOut.Busy,
    Error => ResetOut.Error,
    ErrorID => ResetOut.ErrorID); // MC_Reset
ResetOut.Done := Reset.Done;
END_ACTION

END_FUNCTION_BLOCK

// ---- POUs/POP/FB_LinearActuator_Elec.TcPOU
FUNCTION_BLOCK FB_LinearActuator_Elec EXTENDS FB_BaseDevice IMPLEMENTS I_Device

VAR
	// Instantiation config variables
	nStroke: INT;
	nLead: INT;
	nAccelMax: INT;			// mm/s2
	nVelocityMax: INT; 		// mm/s
	nVelocityJog: INT;		// mm/s
	tExtend: TIME;			// Target time for extend action
	tRetract: TIME;			// Target timef ro retract action
	
	// Motion control variables
	nVelocityExtend: INT;
	nVelocityRetract: INT := 1500;
	
	// Calibration position variables
	nPosExtend: DINT := 75;
	nPosRetract: DINT := 0; 	// (write a fuinction to determine these position limits)
	
	// Motion control function blocks
	mcAxis: 			AXIS_REF;
	//eSMState:			eMoveState;
	
	//eSMState:			eMoveState;
	eSMState: (INIT, ENABLE, EXTEND, EXTEND_SLOW, RETRACT, RETRACT_SLOW, STOP, ERROR, RESET) := INIT;
	
	mcPower: 			MC_Power;
	mcPower_Outputs:	ST_McOutputs;
	
	mcReset: 			MC_Reset;
	mcReset_Outputs:	ST_McOutputs;
	
	mcStop:				MC_Stop;
	mcStop_Outputs:		ST_McOutputs;
	
	mcMoveAbs: 			MC_MoveAbsolute;
	mcMoveAbs_Outputs: 	ST_McOutputs;
	
	mcMoveRel: 			MC_MoveRelative;
	mcMoveRel_Outputs: 	ST_McOutputs;
	
	mcHome:				MC_Home;
	mcHome_Outputs:		ST_McOutputs;
	
	
	tgExecute: R_TRIG;
	tTimeout:	TIME := T#5S;
	fbTON_Timeout: TON := (PT := tTimeout, IN := FALSE);
END_VAR


VAR_INPUT
	bExecute: BOOL := FALSE;
	eMoveType: E_LinActuatorMoveType;
	fbSwitchExtend_1:  FB_AutoSwitch;
	fbSwitchRetract_1: FB_AutoSwitch;
	fbSwitchExtend_2:  FB_AutoSwitch;
	fbSwitchRetract_2: FB_AutoSwitch;
END_VAR

VAR_OUTPUT
	nErrorID: INT;
	bDone: BOOL := FALSE;
END_VAR

(* update the axis status at the beginning of each cycle *)
mcAxis();
tgExecute(CLK := bExecute);
fbTON_Timeout(PT := tTimeout);

// IF eStateTarget <> eState AND (((NOT bExecute) AND bEnable) OR eMode = E_DeviceMode.MANUAL) THEN
IF eStateTarget <> eState AND bEnable OR eMode = E_DeviceMode.MANUAL THEN
	bExecute := TRUE;  // be execute is set to false during movements (allowing a midway change), this behaviour can be stopped if we set bExecite to false after the move is finished
	CASE eStateTarget OF 
		E_DeviceState.EXTENDED:
			eMoveType := E_LinActuatorMoveType.EXTEND;
		E_DeviceState.RETRACTED:
			eMoveType := E_LinActuatorMoveType.RETRACT;
		E_DeviceState.IDLE:
			eMoveType := E_LinActuatorMoveType.STOP;
	END_CASE
END_IF




(* move axis using a state machine *)
CASE eSMState OF

	INIT :	(* initialisation *)
		(* initialize all function blocks *)
		mcMoveAbs.Execute := FALSE;
		mcReset.Execute := FALSE;
		eSMState := ENABLE;

	ENABLE :
		mcPower.Enable := TRUE;
		mcPower.Enable_Positive := TRUE;
		mcPower.Enable_Negative := TRUE;
		IF tgExecute.Q THEN
			fbTON_Timeout.IN := TRUE;
			CASE eMoveType OF
				E_LinActuatorMoveType.EXTEND:
					eSMState := EXTEND;
				E_LinActuatorMoveType.EXTEND_SLOW:
					eSMState := EXTEND_SLOW;
				E_LinActuatorMoveType.RETRACT:
					eSMState := RETRACT;
				E_LinActuatorMoveType.RETRACT_SLOW:
					eSMState := RETRACT_SLOW;
				E_LinActuatorMoveType.STOP:
					eSMState := STOP;
			END_CASE						
		ELSIF mcPower.Error THEN
			eSMState := ERROR;
		END_IF
		
		fbTON_Timeout.IN := FALSE;

	EXTEND :
		eState := E_DeviceState.EXTENDING;							
		mcMoveAbs.Position := nPosExtend;				
		mcMoveAbs.Velocity := nVelocityExtend;			
		mcMoveAbs.BufferMode := MC_Buffered;
		mcMoveAbs.Execute := TRUE;
		IF mcMoveAbs.Done AND (fbSwitchExtend_1.getState() = E_DeviceState.ON AND fbSwitchExtend_2.getState() = E_DeviceState.ON) THEN
			mcMoveAbs.Execute := FALSE;
			eState := E_DeviceState.EXTENDED;
			eSMState := ENABLE;
		ELSIF mcMoveAbs.CommandAborted OR mcMoveAbs.Error OR fbTON_Timeout.Q THEN
			eSMState := ERROR;
		END_IF
		bExecute := FALSE;

	EXTEND_SLOW :				
		eState := E_DeviceState.EXTENDING;			
		mcMoveAbs.Position := nPosExtend;				
		mcMoveAbs.Velocity := nVelocityJog;			
		mcMoveAbs.BufferMode := MC_Buffered;
		mcMoveAbs.Execute := TRUE;
		IF mcMoveAbs.Done AND (fbSwitchExtend_1.getState() = E_DeviceState.ON AND fbSwitchExtend_2.getState() = E_DeviceState.ON) THEN
			eState := E_DeviceState.EXTENDED;
			mcMoveAbs.Execute := FALSE;
			eSMState := ENABLE;
		ELSIF mcMoveAbs.CommandAborted OR mcMoveAbs.Error OR fbTON_Timeout.Q THEN
			eSMState := ERROR;
		END_IF		
		bExecute := FALSE;
		
	RETRACT :			
		eState := E_DeviceState.RETRACTING;	
		
		mcMoveRel.Distance := -20000;
		mcMoveRel.Velocity := 2000;
		mcMoveRel.BufferMode := MC_Buffered;
		mcMoveRel.Execute := TRUE;
		
		IF mcMoveRel.Done THEN // AND (fbSwitchRetract_1.getState() = E_DeviceState.ON AND fbSwitchRetract_2.getState() = E_DeviceState.ON) THEN
			eState := E_DeviceState.RETRACTED;
			mcMoveAbs.Execute := FALSE;
			eSMState := ENABLE;
		ELSIF mcMoveAbs.CommandAborted OR mcMoveAbs.Error OR fbTON_Timeout.Q THEN
			eSMState := ERROR;
		END_IF
		bExecute := FALSE;
		
		
		(*
		mcMoveAbs.Position := nPosRetract;				
		mcMoveAbs.Velocity := nVelocityRetract;			
		mcMoveAbs.BufferMode := MC_Buffered;
		mcMoveAbs.Execute := TRUE;
		IF mcMoveAbs.Done AND (fbSwitchRetract_1.getState() = E_DeviceState.ON AND fbSwitchRetract_2.getState() = E_DeviceState.ON) THEN
			eState := E_DeviceState.RETRACTED;
			mcMoveAbs.Execute := FALSE;
			eSMState := ENABLE;
		ELSIF mcMoveAbs.CommandAborted OR mcMoveAbs.Error OR fbTON_Timeout.Q THEN
			eSMState := ERROR;
		END_IF
		bExecute := FALSE;
		*)

	RETRACT_SLOW :					
		eState := E_DeviceState.RETRACTING;		
		mcMoveAbs.Position := nPosRetract;				
		mcMoveAbs.Velocity := nVelocityJog;			
		mcMoveAbs.BufferMode := MC_Buffered;
		mcMoveAbs.Execute := TRUE;
		IF mcMoveAbs.Done AND (fbSwitchRetract_1.getState() = E_DeviceState.ON AND fbSwitchRetract_2.getState() = E_DeviceState.ON) THEN
			eState := E_DeviceState.RETRACTED;
			mcMoveAbs.Execute := FALSE;
			eSMState := ENABLE;
		ELSIF mcMoveAbs.CommandAborted OR mcMoveAbs.Error OR fbTON_Timeout.Q THEN
			eSMState := ERROR;
		END_IF		
		bExecute := FALSE;
		
	STOP :
		mcStop.Execute := TRUE;
		IF mcStop.Done THEN
			mcStop.Execute := FALSE;
			eSMState := ENABLE;
		END_IF


	ERROR :
		IF mcAxis.Status.Error THEN
			eSMState := RESET;			(* axis error requires reset *)
		ELSIF fbTON_Timeout.Q THEN
			// Raise an alarm that the auto switch was not reached
		ELSE
			eSMState := INIT;			(* function block errors don't need a reset *)
		END_IF
		

	RESET :
		mcReset.Execute := TRUE;
		IF mcReset.Done THEN
			eSMState := INIT;
		ELSIF mcReset.Error THEN
			eSMState := INIT; 			(* can't do anything here *)
		END_IF

END_CASE




// Execute the motion control function blocks 
mcPower(Axis := mcAxis, 
		Enable := mcPower.Enable, 
		Enable_Positive := mcPower.Enable_Positive, 
		Enable_Negative := mcPower.Enable_Negative, 
		Override := 100, 
		Status => mcPower_Outputs.Done, 
		Busy => mcPower_Outputs.Busy, 
		Active => mcPower_Outputs.Active, 
		Error => mcPower_Outputs.Error, 
		ErrorID => mcPower_Outputs.ErrorID);


mcMoveAbs(Axis := mcAxis,
			Execute := mcMoveAbs.Execute,
			Position := mcMoveAbs.Position,
			Velocity := mcMoveAbs.Velocity,
			BufferMode := mcMoveAbs.BufferMode,
			Done => mcMoveAbs_Outputs.Done,
			Busy => mcMoveAbs_Outputs.Busy,
			Active => mcMoveAbs_Outputs.Active,
			CommandAborted => mcMoveAbs_Outputs.CommandAborted,
			Error => mcMoveAbs_Outputs.Error,
			ErrorID => mcMoveAbs_Outputs.ErrorID);
			
mcMoveRel(Axis := mcAxis,
			Execute := mcMoveRel.Execute,
			Distance := mcMoveRel.Distance,
			Velocity := mcMoveRel.Velocity,
			BufferMode := mcMoveRel.BufferMode,
			Busy => mcMoveRel_Outputs.Busy,
			Active => mcMoveRel_Outputs.Active,
			CommandAborted => mcMoveRel_Outputs.CommandAborted,
			Error => mcMoveRel_Outputs.Error,
			ErrorID => mcMoveRel_Outputs.ErrorID);
			
			
mcReset(Axis := mcAxis,
		Execute := mcReset.Execute,
		Done => mcReset_Outputs.Done,
		Busy => mcReset_Outputs.Busy,
		Error => mcReset_Outputs.Error,
		ErrorID => mcReset_Outputs.ErrorID);
		
mcStop(Axis := mcAxis,
		Execute := mcStop.Execute,
		Done => mcStop_Outputs.Done,
		Busy => mcStop_Outputs.Busy,
		Active => mcStop_Outputs.Active,
		CommandAborted => mcStop_Outputs.CommandAborted,
		Error => mcStop_Outputs.Error,
		ErrorId => mcStop_Outputs.ErrorID);

mcHome(Axis := mcAxis,
		Execute := mcHome.Execute,
		Done => mcHome_Outputs.Done,
		Busy => mcHome_Outputs.Busy,
		Active => mcHome_Outputs.Active,
		CommandAborted => mcHome_Outputs.CommandAborted,
		Error => mcHome_Outputs.Error,
		ErrorID => mcHome_Outputs.ErrorID);

METHOD calcVels : BOOL
VAR_INPUT
END_VAR
nVelocityExtend := nStroke / (TIME_TO_INT(tExtend)/1000);
nVelocityRetract := nStroke / (TIME_TO_INT(tRetract)/1000);
END_METHOD

METHOD FB_init : BOOL
VAR_INPUT
	bInitRetains : BOOL; // if TRUE, the retain variables are initialized (warm start / cold start)
	bInCopyCode : BOOL;  // if TRUE, the instance afterwards gets moved into the copy code (online change)
	
	Stroke: INT;
	Lead: INT;
	AccelMax: INT;
	VelocityMax: INT;
	VelocityJog: INT;
	TimeExtend: TIME;
	TimeRetract: TIME;
	
	
END_VAR
nStroke := Stroke;
nLead := Lead;
nAccelMax := AccelMax;
nVelocityMax := VelocityMax;
nVelocityJog := VelocityJog;
tExtend := TimeExtend;
tRetract := TimeRetract;

calcVels(); // calculate extend and retract velocities based on the specified action durations
END_METHOD

END_FUNCTION_BLOCK

// ---- POUs/POP/FB_LinearActuator_Pneumatic.TcPOU
FUNCTION_BLOCK FB_LinearActuator_Pneumatic EXTENDS FB_BaseDevice IMPLEMENTS I_Device

VAR
	// Instantiation config variables
	nStroke: INT;
	nAccelMax: INT;			// mm/s2
	nVelocityMax: INT; 		// mm/s
	tExtend: TIME;			// Target time for extend action
	tRetract: TIME;			// Target timef ro retract action
	
	//Output variables
	bOutput_Extend AT %Q*: BOOL;
	bOutput_Retract AT %Q*: BOOL;

	//eSMState:			eMoveState;
	eSMState: (WAIT, EXTEND, RETRACT, STOP, ERROR, RESET) := WAIT;

	tgExecute: 				R_TRIG;
	tTimeout:				TIME := T#3S;
	fbTON_Timeout: TON := 	(PT := tTimeout, IN := FALSE);
END_VAR


VAR_INPUT
	bExecute: BOOL := FALSE;
	eMoveType: E_LinActuatorMoveType;
	fbSwitchExtend:  FB_AutoSwitch;
	fbSwitchRetract: FB_AutoSwitch;
END_VAR

